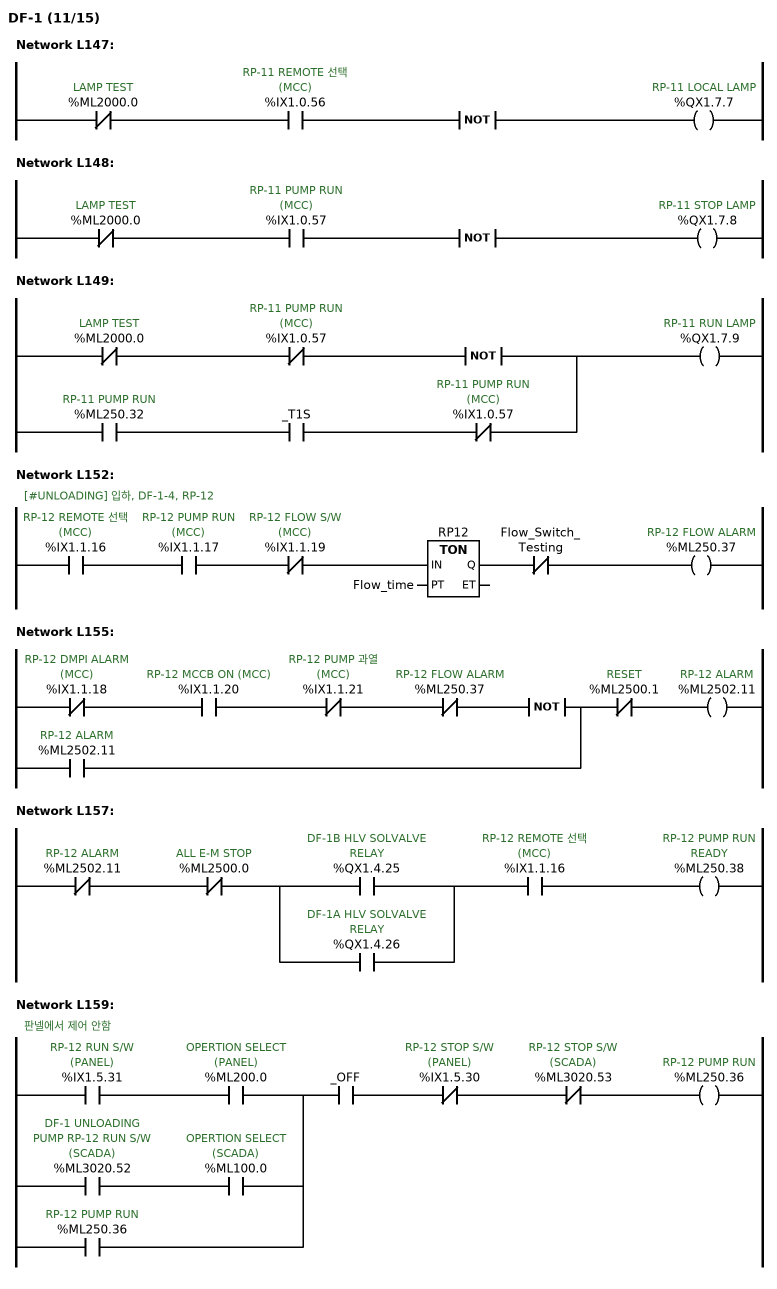
(* Rung L147 *)
%QX1.7.7 := NOT (NOT %ML2000.0 AND %IX1.0.56);
(* Rung L148 *)
%QX1.7.8 := NOT (NOT %ML2000.0 AND %IX1.0.57);
(* Rung L149 *)
%QX1.7.9 := NOT (NOT %ML2000.0 AND NOT %IX1.0.57) OR (%ML250.32 AND _T1S AND NOT %IX1.0.57);
(* [#UNLOADING] 입하, DF-1-4, RP-12 *)
(* Rung L152 *)
RP12(IN := %IX1.1.16 AND %IX1.1.17 AND NOT %IX1.1.19, PT := Flow_time);
%ML250.37 := RP12.Q AND NOT Flow_Switch_Testing;
(* Rung L155 *)
%ML2502.11 := (NOT (NOT %IX1.1.18 AND %IX1.1.20 AND NOT %IX1.1.21 AND NOT %ML250.37) OR %ML2502.11) AND NOT %ML2500.1;
(* Rung L157 *)
%ML250.38 := NOT %ML2502.11 AND NOT %ML2500.0 AND (%QX1.4.25 OR %QX1.4.26) AND %IX1.1.16;
(* Rung L159 *)
%ML250.36 := ((%IX1.5.31 AND %ML200.0) OR (%ML3020.52 AND %ML100.0) OR %ML250.36) AND _OFF AND NOT %IX1.5.30 AND NOT %ML3020.53;
(* 판넬에서 제어 안함 *)

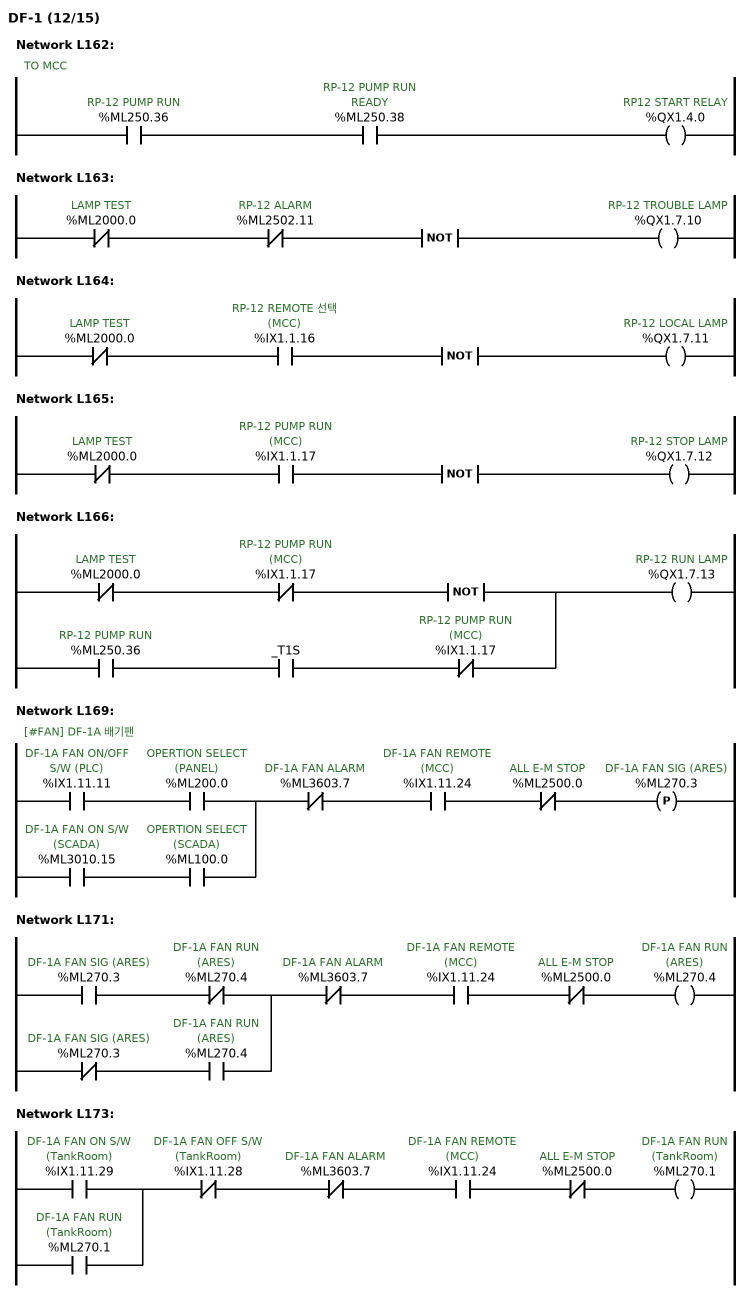
(* Rung L162 *)
%QX1.4.0 := %ML250.36 AND %ML250.38;
(* TO MCC *)
(* Rung L163 *)
%QX1.7.10 := NOT (NOT %ML2000.0 AND NOT %ML2502.11);
(* Rung L164 *)
%QX1.7.11 := NOT (NOT %ML2000.0 AND %IX1.1.16);
(* Rung L165 *)
%QX1.7.12 := NOT (NOT %ML2000.0 AND %IX1.1.17);
(* Rung L166 *)
%QX1.7.13 := NOT (NOT %ML2000.0 AND NOT %IX1.1.17) OR (%ML250.36 AND _T1S AND NOT %IX1.1.17);
(* [#FAN] DF-1A 배기팬 *)
(* Rung L169 *)
_e1(CLK := ((%IX1.11.11 AND %ML200.0) OR (%ML3010.15 AND %ML100.0)) AND NOT %ML3603.7 AND %IX1.11.24 AND NOT %ML2500.0);
%ML270.3 := _e1.Q;
(* Rung L171 *)
%ML270.4 := ((%ML270.3 AND NOT %ML270.4) OR (NOT %ML270.3 AND %ML270.4)) AND NOT %ML3603.7 AND %IX1.11.24 AND NOT %ML2500.0;
(* Rung L173 *)
%ML270.1 := (%IX1.11.29 OR %ML270.1) AND NOT %IX1.11.28 AND NOT %ML3603.7 AND %IX1.11.24 AND NOT %ML2500.0;

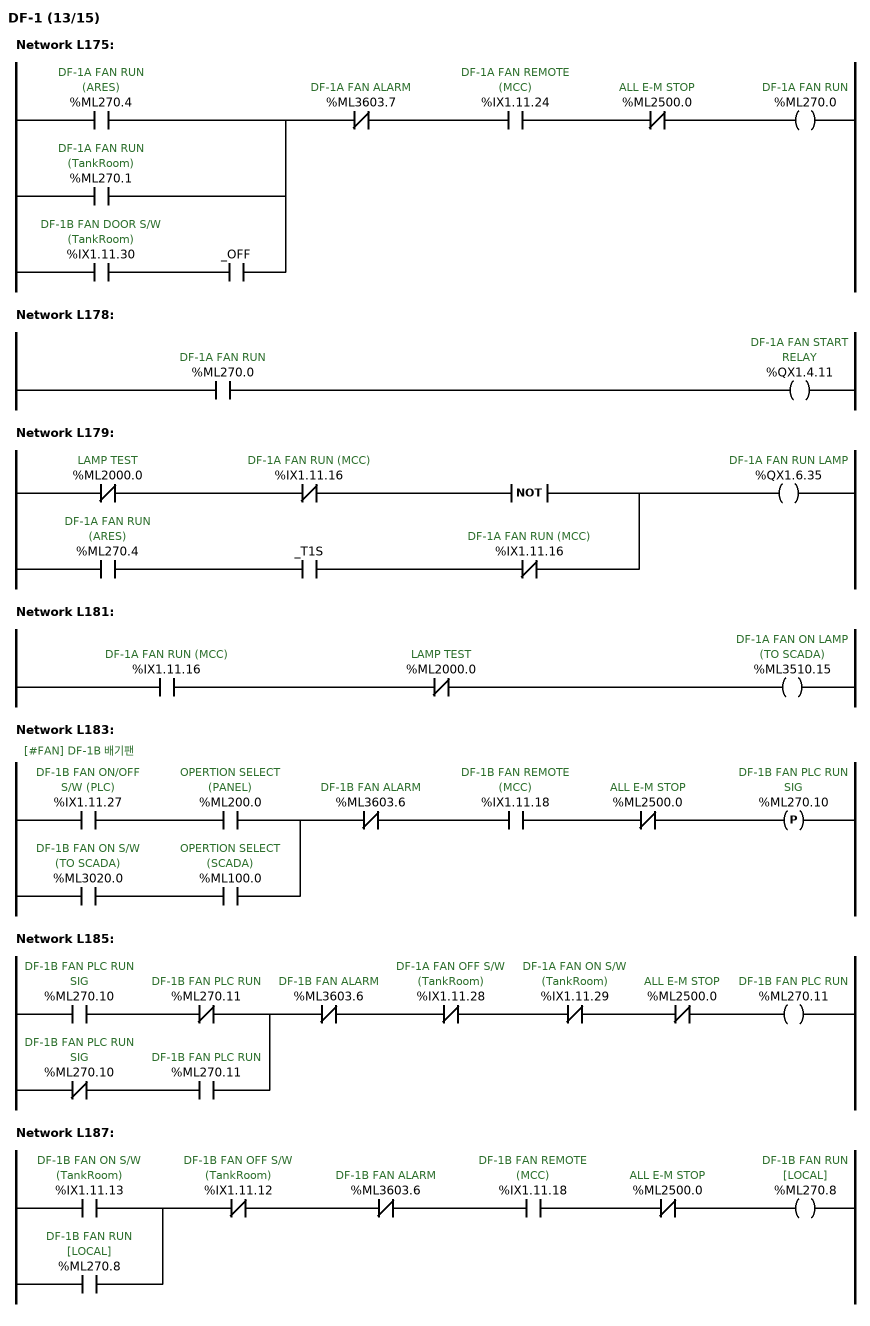
(* Rung L175 *)
%ML270.0 := (%ML270.4 OR %ML270.1 OR (%IX1.11.30 AND _OFF)) AND NOT %ML3603.7 AND %IX1.11.24 AND NOT %ML2500.0;
(* Rung L178 *)
%QX1.4.11 := %ML270.0;
(* Rung L179 *)
%QX1.6.35 := NOT (NOT %ML2000.0 AND NOT %IX1.11.16) OR (%ML270.4 AND _T1S AND NOT %IX1.11.16);
(* Rung L181 *)
%ML3510.15 := %IX1.11.16 AND NOT %ML2000.0;
(* [#FAN] DF-1B 배기팬 *)
(* Rung L183 *)
_e2(CLK := ((%IX1.11.27 AND %ML200.0) OR (%ML3020.0 AND %ML100.0)) AND NOT %ML3603.6 AND %IX1.11.18 AND NOT %ML2500.0);
%ML270.10 := _e2.Q;
(* Rung L185 *)
%ML270.11 := ((%ML270.10 AND NOT %ML270.11) OR (NOT %ML270.10 AND %ML270.11)) AND NOT %ML3603.6 AND NOT %IX1.11.28 AND NOT %IX1.11.29 AND NOT %ML2500.0;
(* Rung L187 *)
%ML270.8 := (%IX1.11.13 OR %ML270.8) AND NOT %IX1.11.12 AND NOT %ML3603.6 AND %IX1.11.18 AND NOT %ML2500.0;

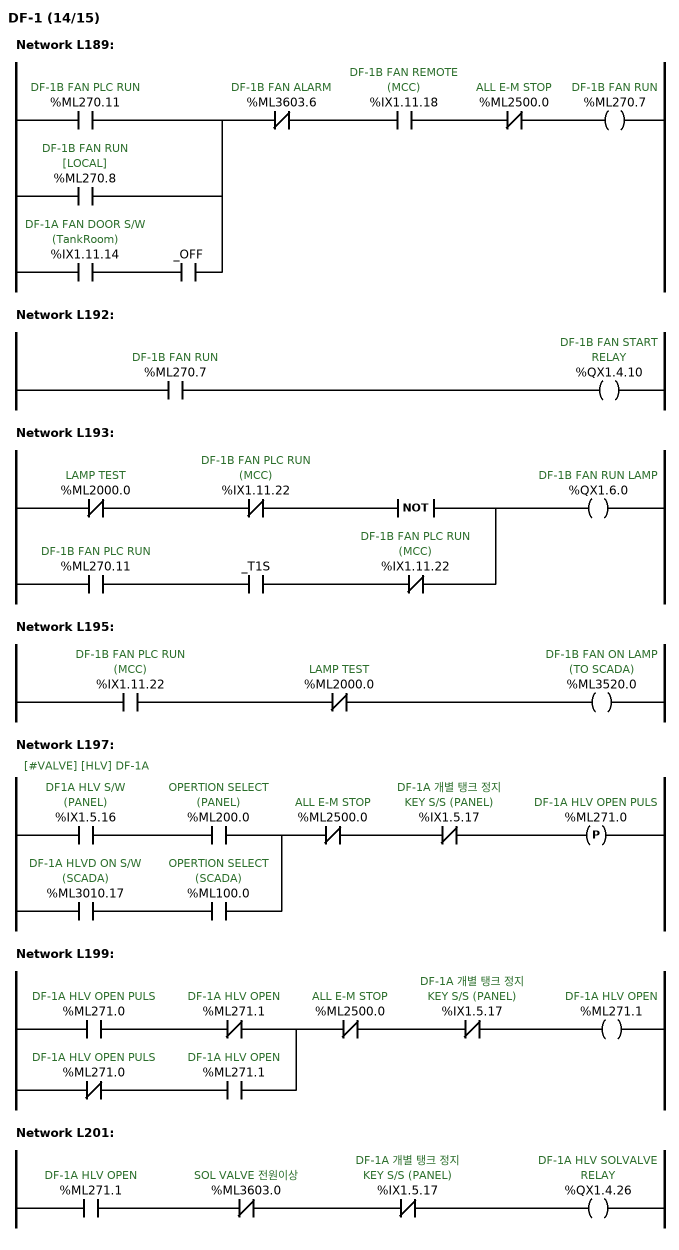
(* Rung L189 *)
%ML270.7 := (%ML270.11 OR %ML270.8 OR (%IX1.11.14 AND _OFF)) AND NOT %ML3603.6 AND %IX1.11.18 AND NOT %ML2500.0;
(* Rung L192 *)
%QX1.4.10 := %ML270.7;
(* Rung L193 *)
%QX1.6.0 := NOT (NOT %ML2000.0 AND NOT %IX1.11.22) OR (%ML270.11 AND _T1S AND NOT %IX1.11.22);
(* Rung L195 *)
%ML3520.0 := %IX1.11.22 AND NOT %ML2000.0;
(* [#VALVE] [HLV] DF-1A *)
(* Rung L197 *)
_e3(CLK := ((%IX1.5.16 AND %ML200.0) OR (%ML3010.17 AND %ML100.0)) AND NOT %ML2500.0 AND NOT %IX1.5.17);
%ML271.0 := _e3.Q;
(* Rung L199 *)
%ML271.1 := ((%ML271.0 AND NOT %ML271.1) OR (NOT %ML271.0 AND %ML271.1)) AND NOT %ML2500.0 AND NOT %IX1.5.17;
(* Rung L201 *)
%QX1.4.26 := %ML271.1 AND NOT %ML3603.0 AND NOT %IX1.5.17;

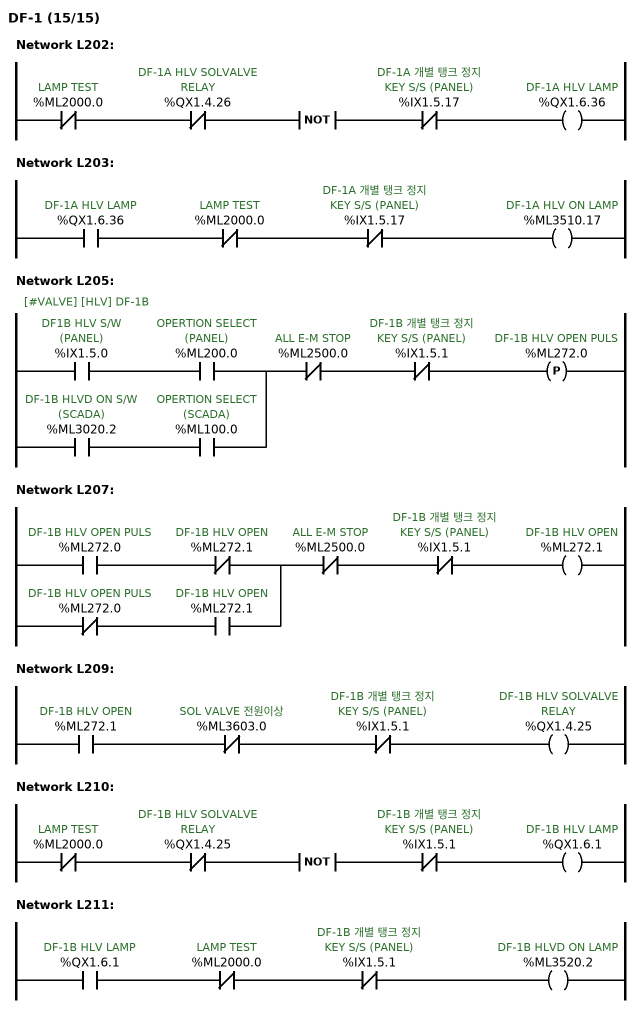
(* Rung L202 *)
%QX1.6.36 := NOT (NOT %ML2000.0 AND NOT %QX1.4.26) AND NOT %IX1.5.17;
(* Rung L203 *)
%ML3510.17 := %QX1.6.36 AND NOT %ML2000.0 AND NOT %IX1.5.17;
(* [#VALVE] [HLV] DF-1B *)
(* Rung L205 *)
_e4(CLK := ((%IX1.5.0 AND %ML200.0) OR (%ML3020.2 AND %ML100.0)) AND NOT %ML2500.0 AND NOT %IX1.5.1);
%ML272.0 := _e4.Q;
(* Rung L207 *)
%ML272.1 := ((%ML272.0 AND NOT %ML272.1) OR (NOT %ML272.0 AND %ML272.1)) AND NOT %ML2500.0 AND NOT %IX1.5.1;
(* Rung L209 *)
%QX1.4.25 := %ML272.1 AND NOT %ML3603.0 AND NOT %IX1.5.1;
(* Rung L210 *)
%QX1.6.1 := NOT (NOT %ML2000.0 AND NOT %QX1.4.25) AND NOT %IX1.5.1;
(* Rung L211 *)
%ML3520.2 := %QX1.6.1 AND NOT %ML2000.0 AND NOT %IX1.5.1;
END_PROGRAM

PROGRAM DF-M (* task: 스캔 프로그램 *)
VAR_EXTERNAL
    Flow_Switch_Testing : BOOL;
    Flow_time : TIME;
END_VAR
VAR
    RP10 : TON;
    RP11 : TON;
    RP12 : TON;
    RP13 : TON;
    RP14 : TON;
    RP15 : TON;
    RP16 : TON;
    RP17 : TON;
    RP18 : TON;
    RP7 : TON;
    RP8 : TON;
    RP9 : TON;
    SUMP02 : TON; (* SP-2 *)
    SUMP04 : TON;
END_VAR
VAR
    _t1 : BOOL;
    _t2 : BOOL;
    _t3 : BOOL;
    _t4 : BOOL;
    _e5 : R_TRIG;
END_VAR

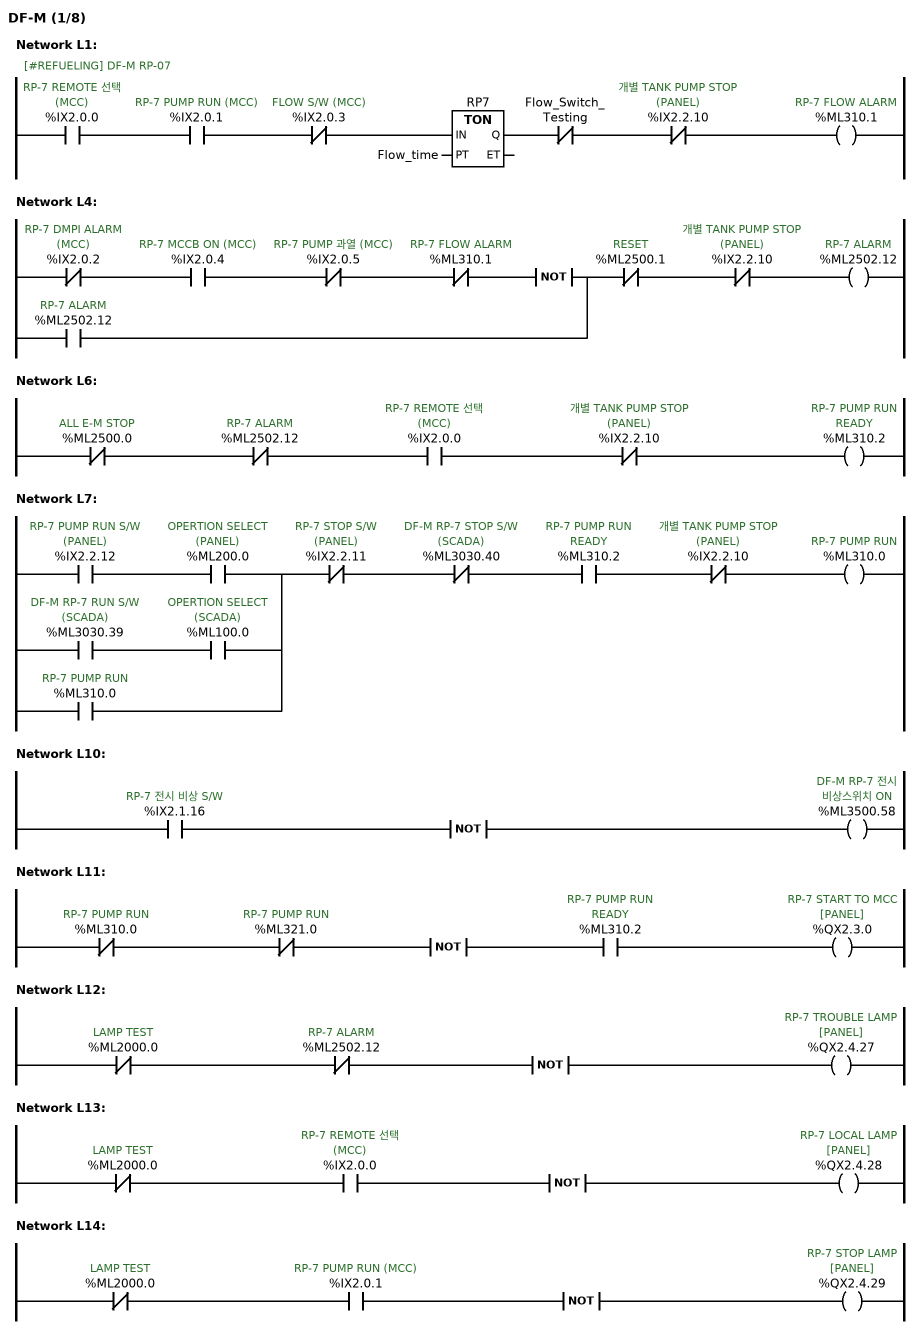
(* [#REFUELING] DF-M RP-07 *)
(* Rung L1 *)
RP7(IN := %IX2.0.0 AND %IX2.0.1 AND NOT %IX2.0.3, PT := Flow_time);
%ML310.1 := RP7.Q AND NOT Flow_Switch_Testing AND NOT %IX2.2.10;
(* Rung L4 *)
%ML2502.12 := (NOT (NOT %IX2.0.2 AND %IX2.0.4 AND NOT %IX2.0.5 AND NOT %ML310.1) OR %ML2502.12) AND NOT %ML2500.1 AND NOT %IX2.2.10;
(* Rung L6 *)
%ML310.2 := NOT %ML2500.0 AND NOT %ML2502.12 AND %IX2.0.0 AND NOT %IX2.2.10;
(* Rung L7 *)
%ML310.0 := ((%IX2.2.12 AND %ML200.0) OR (%ML3030.39 AND %ML100.0) OR %ML310.0) AND NOT %IX2.2.11 AND NOT %ML3030.40 AND %ML310.2 AND NOT %IX2.2.10;
(* Rung L10 *)
%ML3500.58 := NOT %IX2.1.16;
(* Rung L11 *)
%QX2.3.0 := NOT (NOT %ML310.0 AND NOT %ML321.0) AND %ML310.2;
(* Rung L12 *)
%QX2.4.27 := NOT (NOT %ML2000.0 AND NOT %ML2502.12);
(* Rung L13 *)
%QX2.4.28 := NOT (NOT %ML2000.0 AND %IX2.0.0);
(* Rung L14 *)
%QX2.4.29 := NOT (NOT %ML2000.0 AND %IX2.0.1);

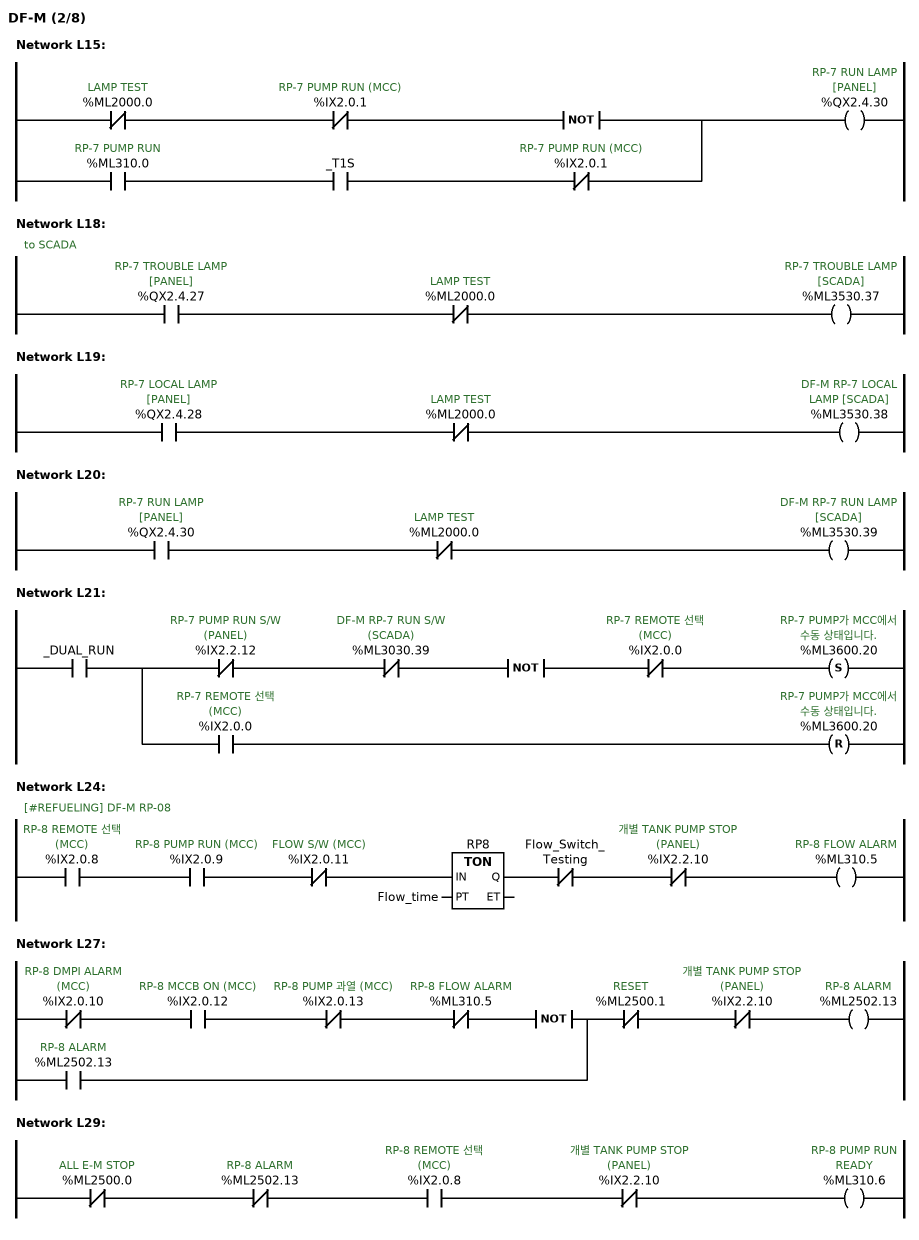
(* Rung L15 *)
%QX2.4.30 := NOT (NOT %ML2000.0 AND NOT %IX2.0.1) OR (%ML310.0 AND _T1S AND NOT %IX2.0.1);
(* to SCADA *)
(* Rung L18 *)
%ML3530.37 := %QX2.4.27 AND NOT %ML2000.0;
(* Rung L19 *)
%ML3530.38 := %QX2.4.28 AND NOT %ML2000.0;
(* Rung L20 *)
%ML3530.39 := %QX2.4.30 AND NOT %ML2000.0;
(* Rung L21 *)
IF NOT (_DUAL_RUN AND NOT %IX2.2.12 AND NOT %ML3030.39) AND NOT %IX2.0.0 THEN %ML3600.20 := TRUE; END_IF;
IF _DUAL_RUN AND %IX2.0.0 THEN %ML3600.20 := FALSE; END_IF;
(* [#REFUELING] DF-M RP-08 *)
(* Rung L24 *)
RP8(IN := %IX2.0.8 AND %IX2.0.9 AND NOT %IX2.0.11, PT := Flow_time);
%ML310.5 := RP8.Q AND NOT Flow_Switch_Testing AND NOT %IX2.2.10;
(* Rung L27 *)
%ML2502.13 := (NOT (NOT %IX2.0.10 AND %IX2.0.12 AND NOT %IX2.0.13 AND NOT %ML310.5) OR %ML2502.13) AND NOT %ML2500.1 AND NOT %IX2.2.10;
(* Rung L29 *)
%ML310.6 := NOT %ML2500.0 AND NOT %ML2502.13 AND %IX2.0.8 AND NOT %IX2.2.10;

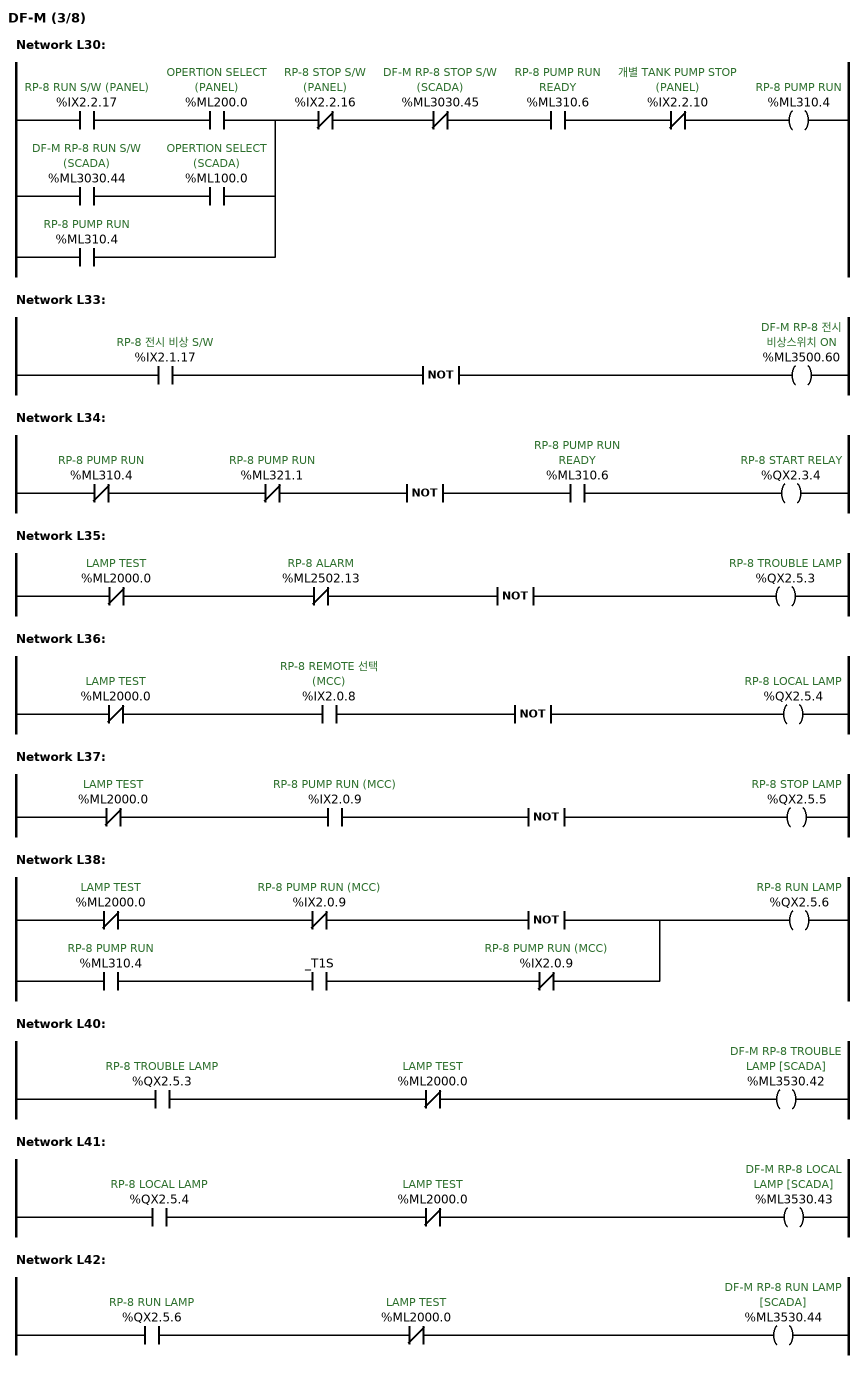
(* Rung L30 *)
%ML310.4 := ((%IX2.2.17 AND %ML200.0) OR (%ML3030.44 AND %ML100.0) OR %ML310.4) AND NOT %IX2.2.16 AND NOT %ML3030.45 AND %ML310.6 AND NOT %IX2.2.10;
(* Rung L33 *)
%ML3500.60 := NOT %IX2.1.17;
(* Rung L34 *)
%QX2.3.4 := NOT (NOT %ML310.4 AND NOT %ML321.1) AND %ML310.6;
(* Rung L35 *)
%QX2.5.3 := NOT (NOT %ML2000.0 AND NOT %ML2502.13);
(* Rung L36 *)
%QX2.5.4 := NOT (NOT %ML2000.0 AND %IX2.0.8);
(* Rung L37 *)
%QX2.5.5 := NOT (NOT %ML2000.0 AND %IX2.0.9);
(* Rung L38 *)
%QX2.5.6 := NOT (NOT %ML2000.0 AND NOT %IX2.0.9) OR (%ML310.4 AND _T1S AND NOT %IX2.0.9);
(* Rung L40 *)
%ML3530.42 := %QX2.5.3 AND NOT %ML2000.0;
(* Rung L41 *)
%ML3530.43 := %QX2.5.4 AND NOT %ML2000.0;
(* Rung L42 *)
%ML3530.44 := %QX2.5.6 AND NOT %ML2000.0;

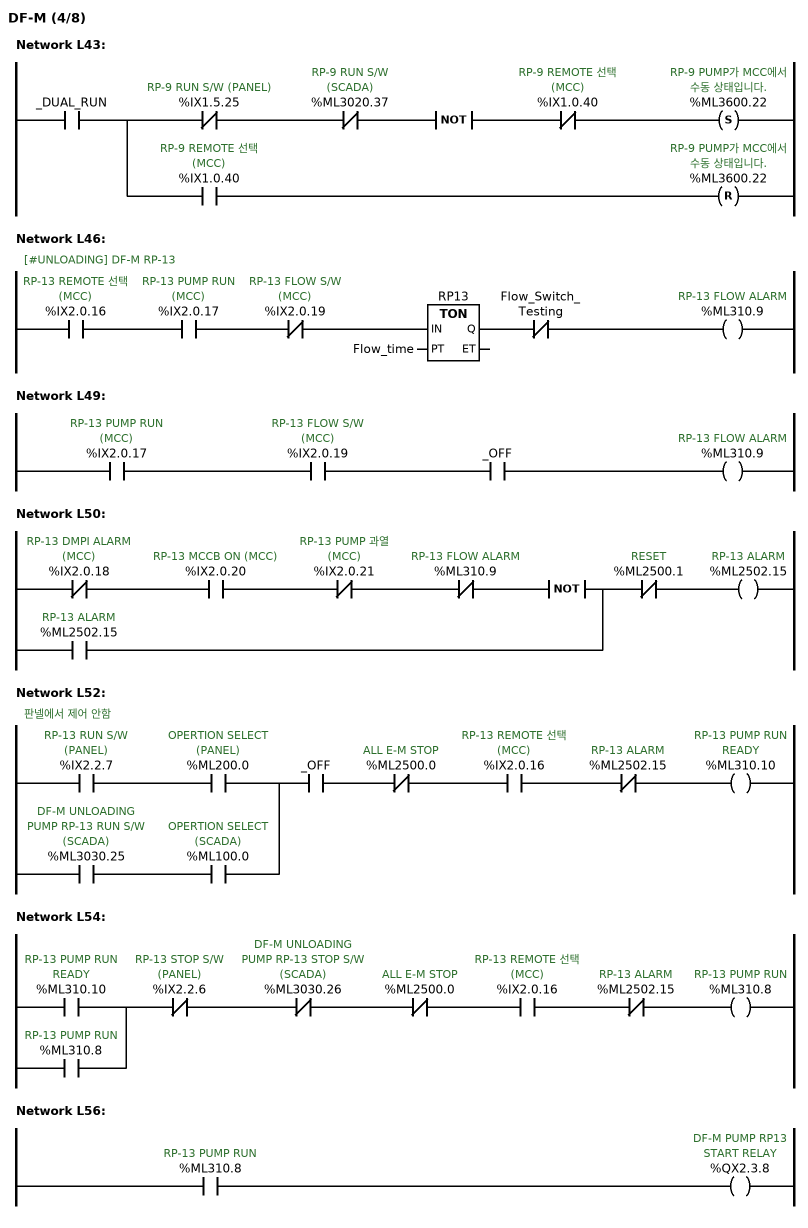
(* Rung L43 *)
IF NOT (_DUAL_RUN AND NOT %IX1.5.25 AND NOT %ML3020.37) AND NOT %IX1.0.40 THEN %ML3600.22 := TRUE; END_IF;
IF _DUAL_RUN AND %IX1.0.40 THEN %ML3600.22 := FALSE; END_IF;
(* [#UNLOADING] DF-M RP-13 *)
(* Rung L46 *)
RP13(IN := %IX2.0.16 AND %IX2.0.17 AND NOT %IX2.0.19, PT := Flow_time);
%ML310.9 := RP13.Q AND NOT Flow_Switch_Testing;
(* Rung L49 *)
%ML310.9 := %IX2.0.17 AND %IX2.0.19 AND _OFF;
(* Rung L50 *)
%ML2502.15 := (NOT (NOT %IX2.0.18 AND %IX2.0.20 AND NOT %IX2.0.21 AND NOT %ML310.9) OR %ML2502.15) AND NOT %ML2500.1;
(* Rung L52 *)
%ML310.10 := ((%IX2.2.7 AND %ML200.0) OR (%ML3030.25 AND %ML100.0)) AND _OFF AND NOT %ML2500.0 AND %IX2.0.16 AND NOT %ML2502.15;
(* 판넬에서 제어 안함 *)
(* Rung L54 *)
%ML310.8 := (%ML310.10 OR %ML310.8) AND NOT %IX2.2.6 AND NOT %ML3030.26 AND NOT %ML2500.0 AND %IX2.0.16 AND NOT %ML2502.15;
(* Rung L56 *)
%QX2.3.8 := %ML310.8;

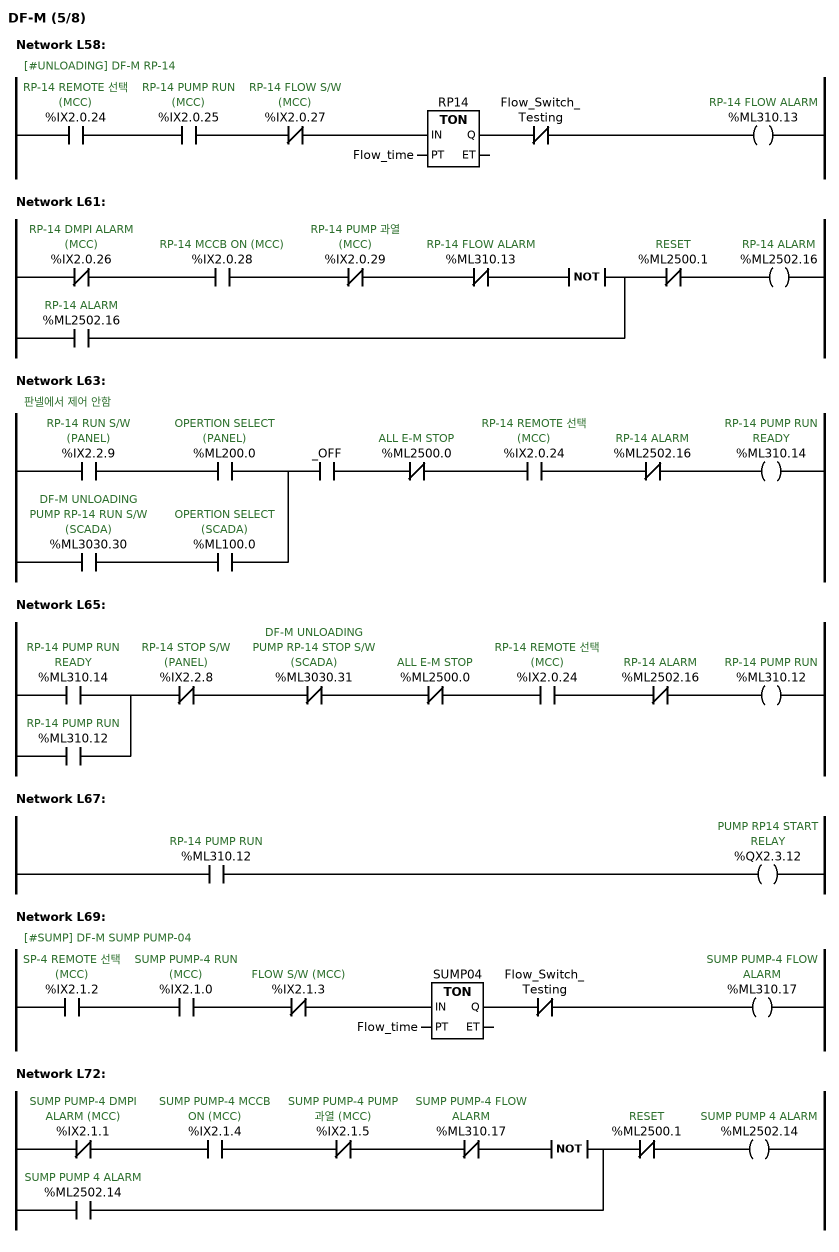
(* [#UNLOADING] DF-M RP-14 *)
(* Rung L58 *)
RP14(IN := %IX2.0.24 AND %IX2.0.25 AND NOT %IX2.0.27, PT := Flow_time);
%ML310.13 := RP14.Q AND NOT Flow_Switch_Testing;
(* Rung L61 *)
%ML2502.16 := (NOT (NOT %IX2.0.26 AND %IX2.0.28 AND NOT %IX2.0.29 AND NOT %ML310.13) OR %ML2502.16) AND NOT %ML2500.1;
(* Rung L63 *)
%ML310.14 := ((%IX2.2.9 AND %ML200.0) OR (%ML3030.30 AND %ML100.0)) AND _OFF AND NOT %ML2500.0 AND %IX2.0.24 AND NOT %ML2502.16;
(* 판넬에서 제어 안함 *)
(* Rung L65 *)
%ML310.12 := (%ML310.14 OR %ML310.12) AND NOT %IX2.2.8 AND NOT %ML3030.31 AND NOT %ML2500.0 AND %IX2.0.24 AND NOT %ML2502.16;
(* Rung L67 *)
%QX2.3.12 := %ML310.12;
(* [#SUMP] DF-M SUMP PUMP-04 *)
(* Rung L69 *)
SUMP04(IN := %IX2.1.2 AND %IX2.1.0 AND NOT %IX2.1.3, PT := Flow_time);
%ML310.17 := SUMP04.Q AND NOT Flow_Switch_Testing;
(* Rung L72 *)
%ML2502.14 := (NOT (NOT %IX2.1.1 AND %IX2.1.4 AND NOT %IX2.1.5 AND NOT %ML310.17) OR %ML2502.14) AND NOT %ML2500.1;

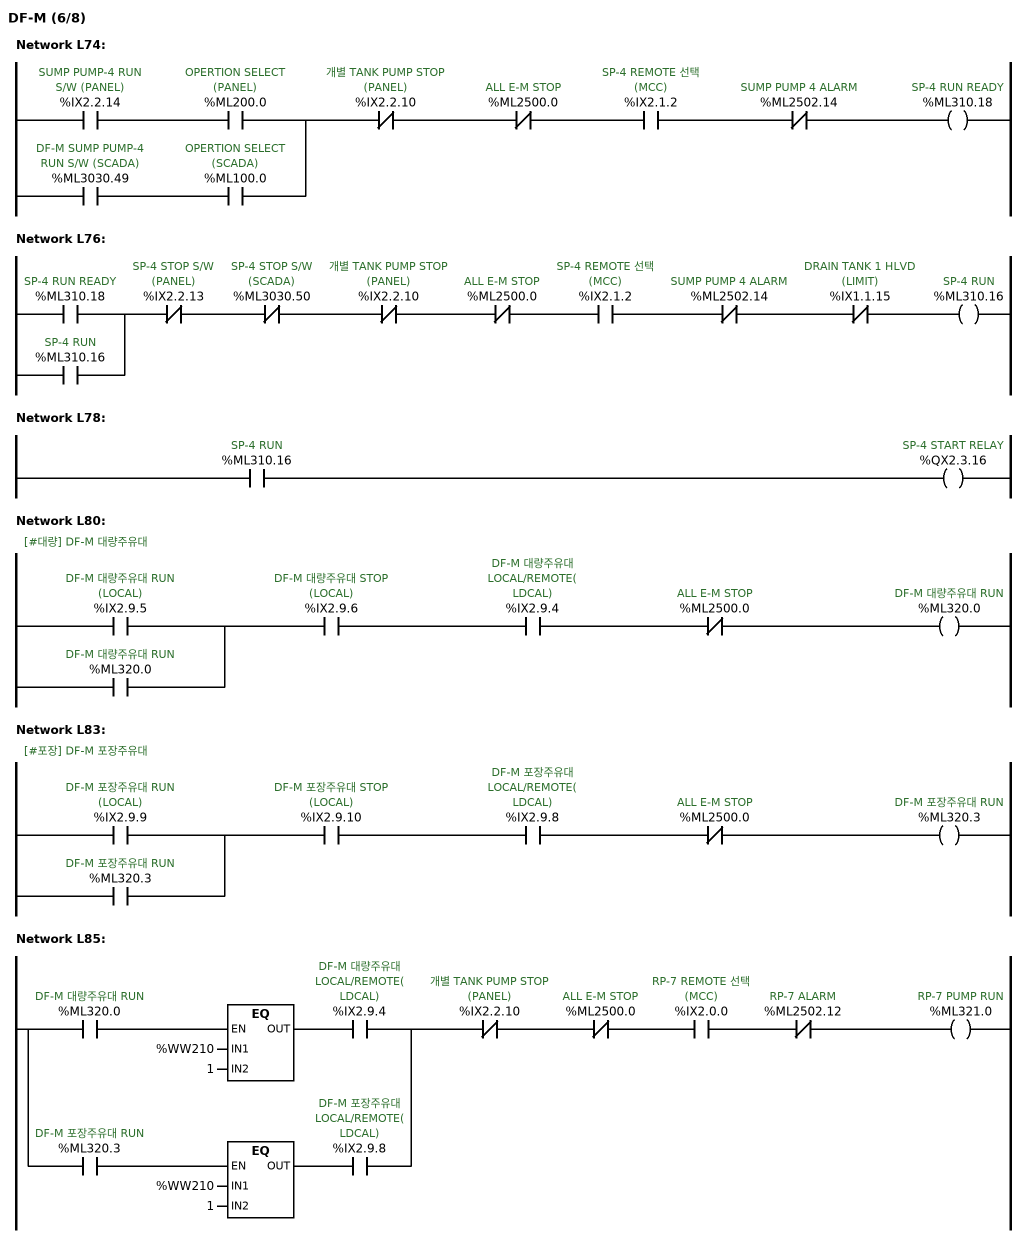
(* Rung L74 *)
%ML310.18 := ((%IX2.2.14 AND %ML200.0) OR (%ML3030.49 AND %ML100.0)) AND NOT %IX2.2.10 AND NOT %ML2500.0 AND %IX2.1.2 AND NOT %ML2502.14;
(* Rung L76 *)
%ML310.16 := (%ML310.18 OR %ML310.16) AND NOT %IX2.2.13 AND NOT %ML3030.50 AND NOT %IX2.2.10 AND NOT %ML2500.0 AND %IX2.1.2 AND NOT %ML2502.14 AND NOT %IX1.1.15;
(* Rung L78 *)
%QX2.3.16 := %ML310.16;
(* [#대량] DF-M 대량주유대 *)
(* Rung L80 *)
%ML320.0 := (%IX2.9.5 OR %ML320.0) AND %IX2.9.6 AND %IX2.9.4 AND NOT %ML2500.0;
(* [#포장] DF-M 포장주유대 *)
(* Rung L83 *)
%ML320.3 := (%IX2.9.9 OR %ML320.3) AND %IX2.9.10 AND %IX2.9.8 AND NOT %ML2500.0;
(* Rung L85 *)
IF %ML320.0 THEN _t1 := %WW210 = 1; END_IF;
IF %ML320.3 THEN _t2 := %WW210 = 1; END_IF;
%ML321.0 := ((_t1 AND %IX2.9.4) OR (_t2 AND %IX2.9.8)) AND NOT %IX2.2.10 AND NOT %ML2500.0 AND %IX2.0.0 AND NOT %ML2502.12;

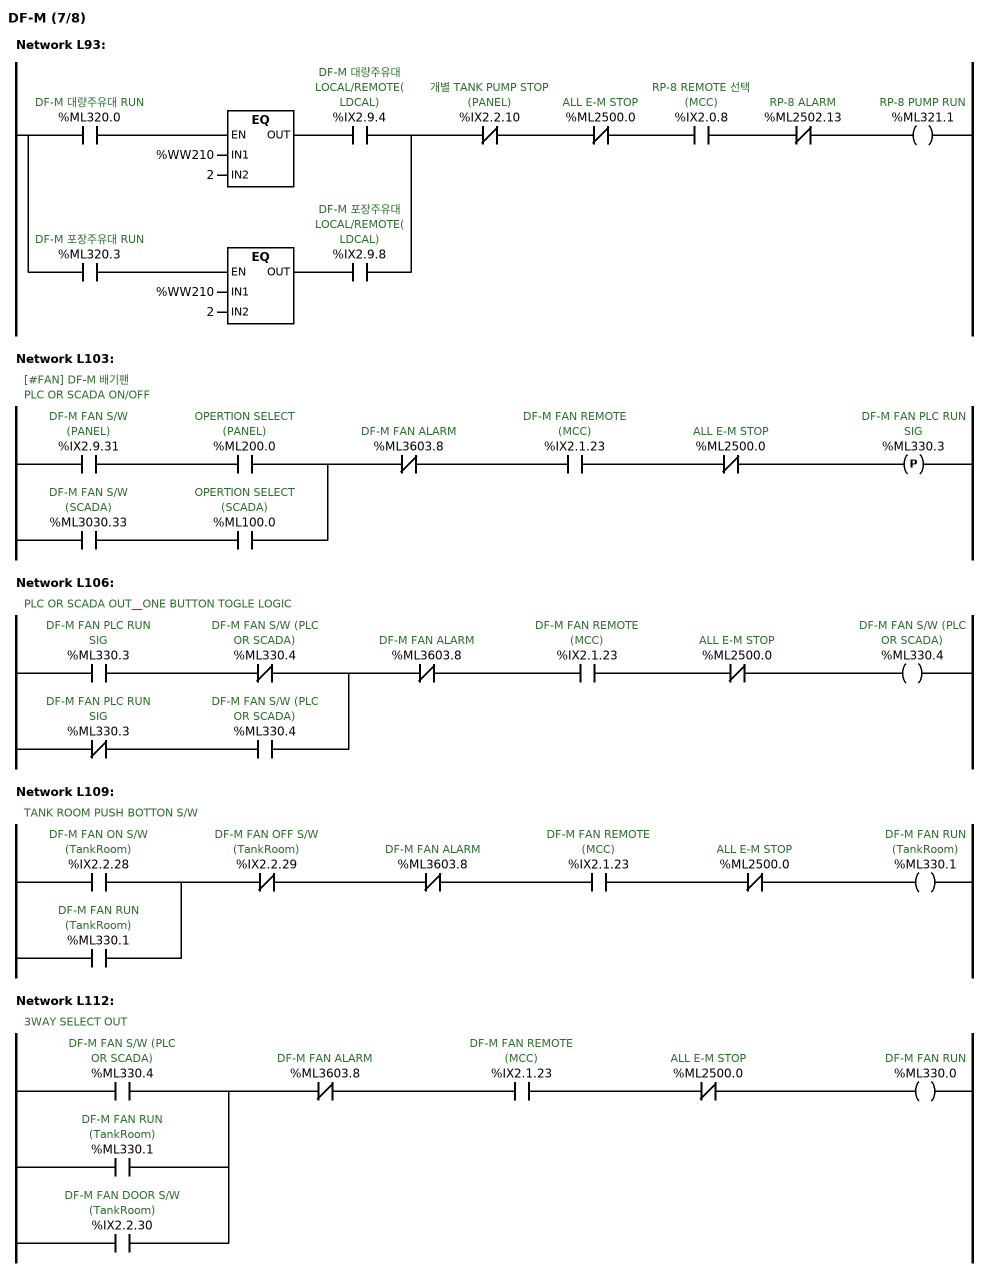
(* Rung L93 *)
IF %ML320.0 THEN _t3 := %WW210 = 2; END_IF;
IF %ML320.3 THEN _t4 := %WW210 = 2; END_IF;
%ML321.1 := ((_t3 AND %IX2.9.4) OR (_t4 AND %IX2.9.8)) AND NOT %IX2.2.10 AND NOT %ML2500.0 AND %IX2.0.8 AND NOT %ML2502.13;
(* [#FAN] DF-M 배기팬 *)
(* PLC OR SCADA ON/OFF *)
(* Rung L103 *)
_e5(CLK := ((%IX2.9.31 AND %ML200.0) OR (%ML3030.33 AND %ML100.0)) AND NOT %ML3603.8 AND %IX2.1.23 AND NOT %ML2500.0);
%ML330.3 := _e5.Q;
(* PLC OR SCADA OUT__ONE BUTTON TOGLE LOGIC *)
(* Rung L106 *)
%ML330.4 := ((%ML330.3 AND NOT %ML330.4) OR (NOT %ML330.3 AND %ML330.4)) AND NOT %ML3603.8 AND %IX2.1.23 AND NOT %ML2500.0;
(* TANK ROOM PUSH BOTTON S/W *)
(* Rung L109 *)
%ML330.1 := (%IX2.2.28 OR %ML330.1) AND NOT %IX2.2.29 AND NOT %ML3603.8 AND %IX2.1.23 AND NOT %ML2500.0;
(* 3WAY SELECT OUT *)
(* Rung L112 *)
%ML330.0 := (%ML330.4 OR %ML330.1 OR %IX2.2.30) AND NOT %ML3603.8 AND %IX2.1.23 AND NOT %ML2500.0;

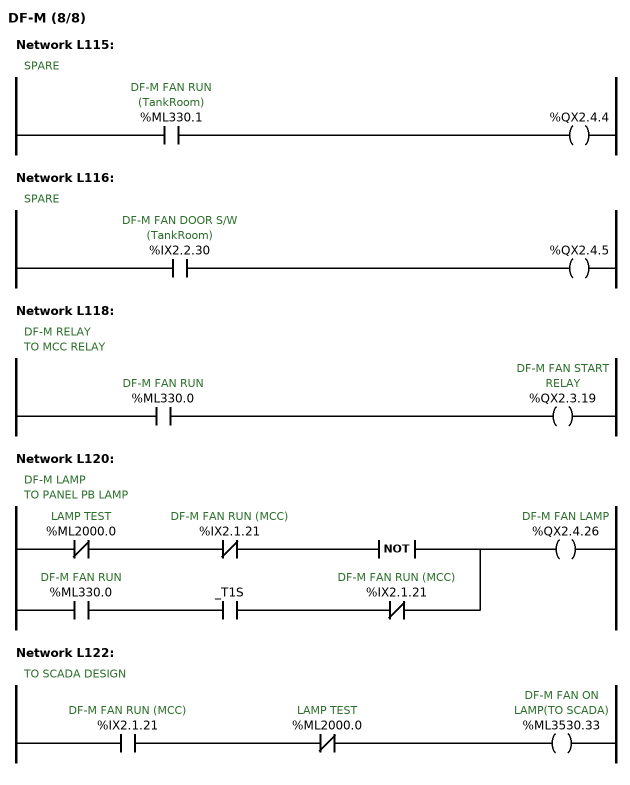
(* Rung L115 *)
%QX2.4.4 := %ML330.1;
(* SPARE *)
(* Rung L116 *)
%QX2.4.5 := %IX2.2.30;
(* SPARE *)
(* DF-M RELAY *)
(* Rung L118 *)
%QX2.3.19 := %ML330.0;
(* TO MCC RELAY *)
(* DF-M LAMP *)
(* Rung L120 *)
%QX2.4.26 := NOT (NOT %ML2000.0 AND NOT %IX2.1.21) OR (%ML330.0 AND _T1S AND NOT %IX2.1.21);
(* TO PANEL PB LAMP *)
(* Rung L122 *)
%ML3530.33 := %IX2.1.21 AND NOT %ML2000.0;
(* TO SCADA DESIGN *)
END_PROGRAM

PROGRAM MOGAS (* task: 스캔 프로그램 *)
VAR
    DP01 : TON; (* DRAIN PUMP FLOW SENSOR *)
    RP10 : TON;
    RP11 : TON;
    RP12 : TON;
    RP13 : TON;
    RP14 : TON;
    RP15 : TON;
    RP16 : TON;
    RP17 : TON;
    RP18 : TON;
    RP19 : TON;
    RP20 : TON;
    RP5 : TON;
    RP6 : TON;
    RP7 : TON;
    RP8 : TON;
    RP9 : TON;
    SUMP04 : TON;
END_VAR
VAR_EXTERNAL
    Flow_Switch_Testing : BOOL;
    Flow_time : TIME;
END_VAR
VAR
    _t1 : BOOL;
    _t2 : BOOL;
    _t3 : BOOL;
    _t4 : BOOL;
    _e5 : R_TRIG;
END_VAR

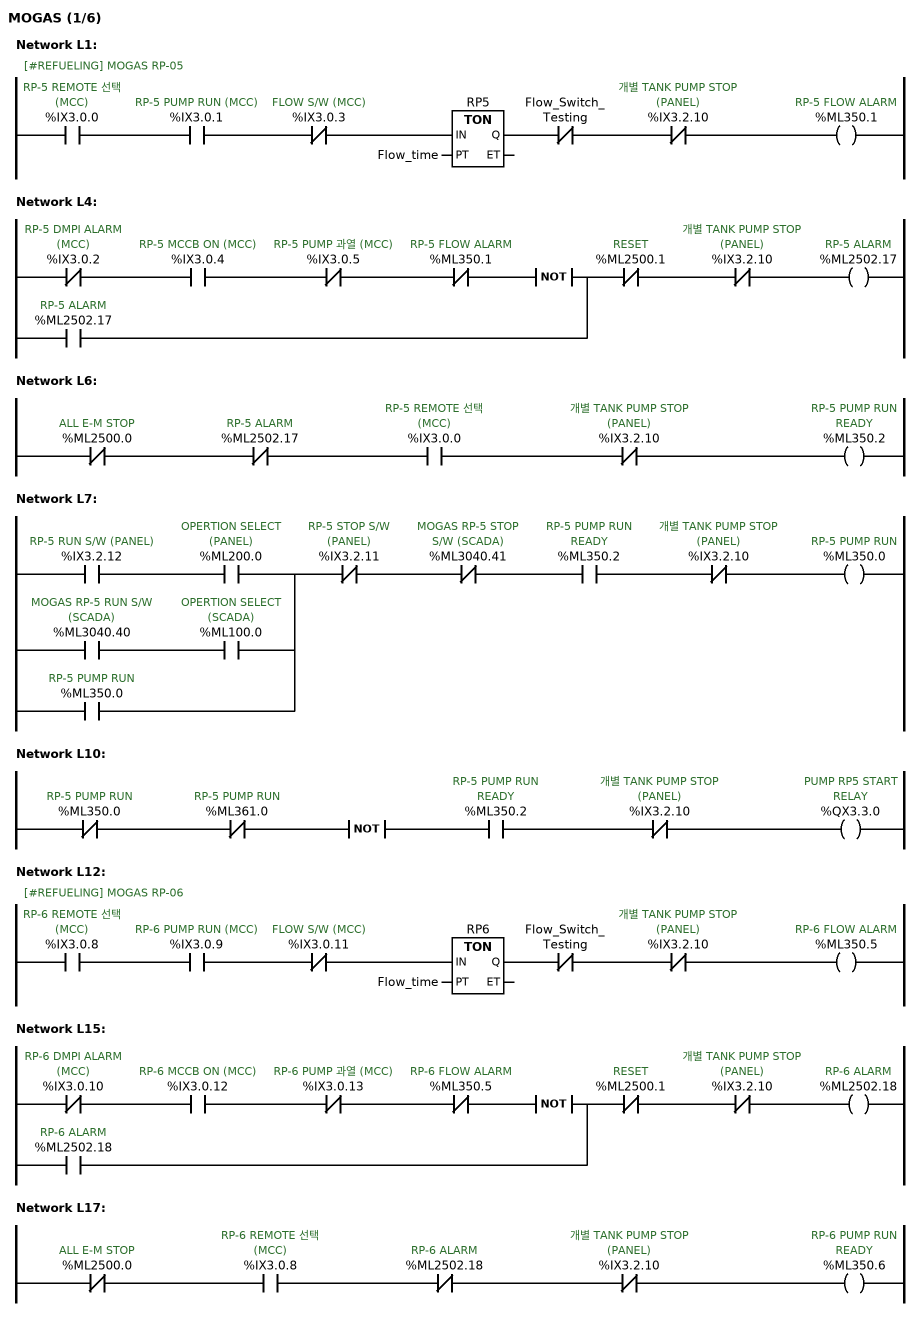
(* [#REFUELING] MOGAS RP-05 *)
(* Rung L1 *)
RP5(IN := %IX3.0.0 AND %IX3.0.1 AND NOT %IX3.0.3, PT := Flow_time);
%ML350.1 := RP5.Q AND NOT Flow_Switch_Testing AND NOT %IX3.2.10;
(* Rung L4 *)
%ML2502.17 := (NOT (NOT %IX3.0.2 AND %IX3.0.4 AND NOT %IX3.0.5 AND NOT %ML350.1) OR %ML2502.17) AND NOT %ML2500.1 AND NOT %IX3.2.10;
(* Rung L6 *)
%ML350.2 := NOT %ML2500.0 AND NOT %ML2502.17 AND %IX3.0.0 AND NOT %IX3.2.10;
(* Rung L7 *)
%ML350.0 := ((%IX3.2.12 AND %ML200.0) OR (%ML3040.40 AND %ML100.0) OR %ML350.0) AND NOT %IX3.2.11 AND NOT %ML3040.41 AND %ML350.2 AND NOT %IX3.2.10;
(* Rung L10 *)
%QX3.3.0 := NOT (NOT %ML350.0 AND NOT %ML361.0) AND %ML350.2 AND NOT %IX3.2.10;
(* [#REFUELING] MOGAS RP-06 *)
(* Rung L12 *)
RP6(IN := %IX3.0.8 AND %IX3.0.9 AND NOT %IX3.0.11, PT := Flow_time);
%ML350.5 := RP6.Q AND NOT Flow_Switch_Testing AND NOT %IX3.2.10;
(* Rung L15 *)
%ML2502.18 := (NOT (NOT %IX3.0.10 AND %IX3.0.12 AND NOT %IX3.0.13 AND NOT %ML350.5) OR %ML2502.18) AND NOT %ML2500.1 AND NOT %IX3.2.10;
(* Rung L17 *)
%ML350.6 := NOT %ML2500.0 AND %IX3.0.8 AND NOT %ML2502.18 AND NOT %IX3.2.10;

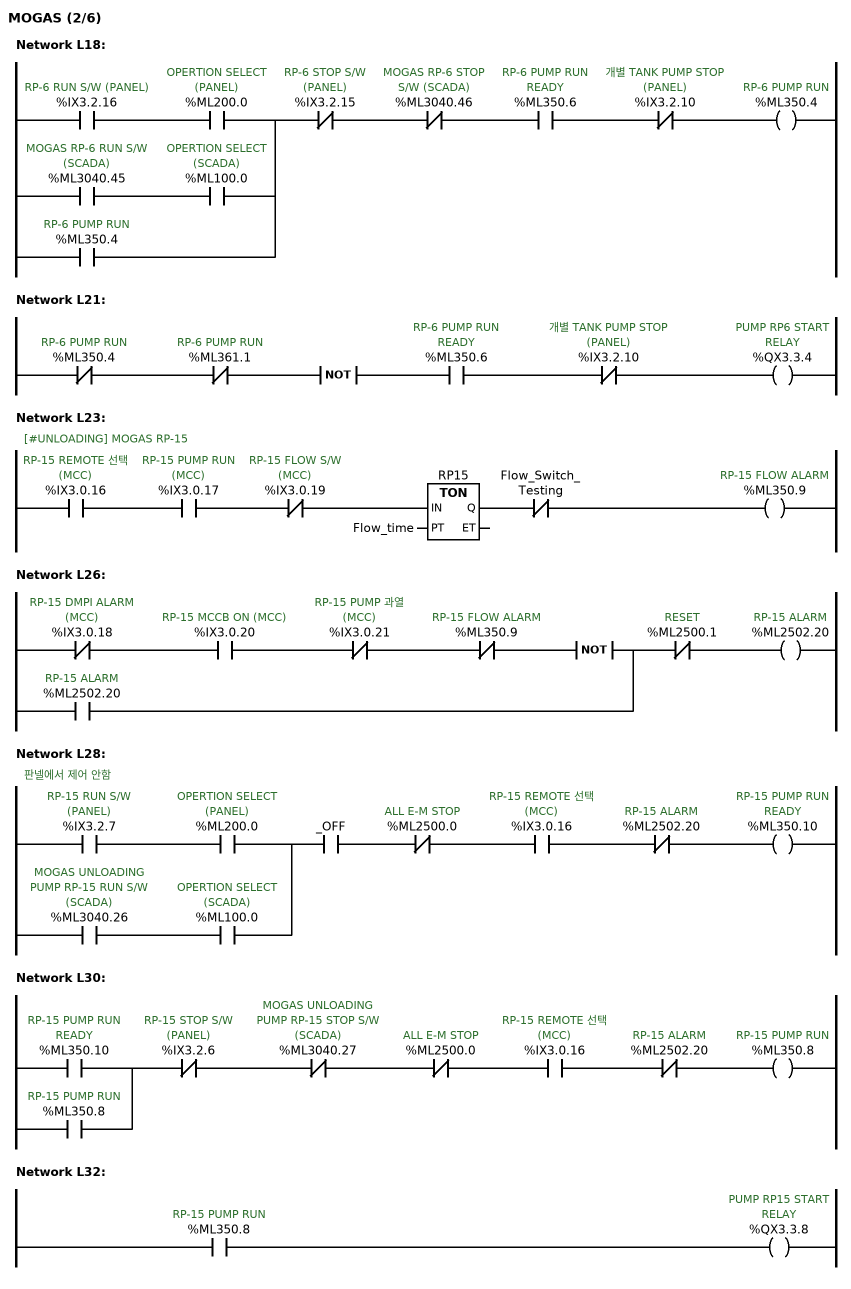
(* Rung L18 *)
%ML350.4 := ((%IX3.2.16 AND %ML200.0) OR (%ML3040.45 AND %ML100.0) OR %ML350.4) AND NOT %IX3.2.15 AND NOT %ML3040.46 AND %ML350.6 AND NOT %IX3.2.10;
(* Rung L21 *)
%QX3.3.4 := NOT (NOT %ML350.4 AND NOT %ML361.1) AND %ML350.6 AND NOT %IX3.2.10;
(* [#UNLOADING] MOGAS RP-15 *)
(* Rung L23 *)
RP15(IN := %IX3.0.16 AND %IX3.0.17 AND NOT %IX3.0.19, PT := Flow_time);
%ML350.9 := RP15.Q AND NOT Flow_Switch_Testing;
(* Rung L26 *)
%ML2502.20 := (NOT (NOT %IX3.0.18 AND %IX3.0.20 AND NOT %IX3.0.21 AND NOT %ML350.9) OR %ML2502.20) AND NOT %ML2500.1;
(* Rung L28 *)
%ML350.10 := ((%IX3.2.7 AND %ML200.0) OR (%ML3040.26 AND %ML100.0)) AND _OFF AND NOT %ML2500.0 AND %IX3.0.16 AND NOT %ML2502.20;
(* 판넬에서 제어 안함 *)
(* Rung L30 *)
%ML350.8 := (%ML350.10 OR %ML350.8) AND NOT %IX3.2.6 AND NOT %ML3040.27 AND NOT %ML2500.0 AND %IX3.0.16 AND NOT %ML2502.20;
(* Rung L32 *)
%QX3.3.8 := %ML350.8;

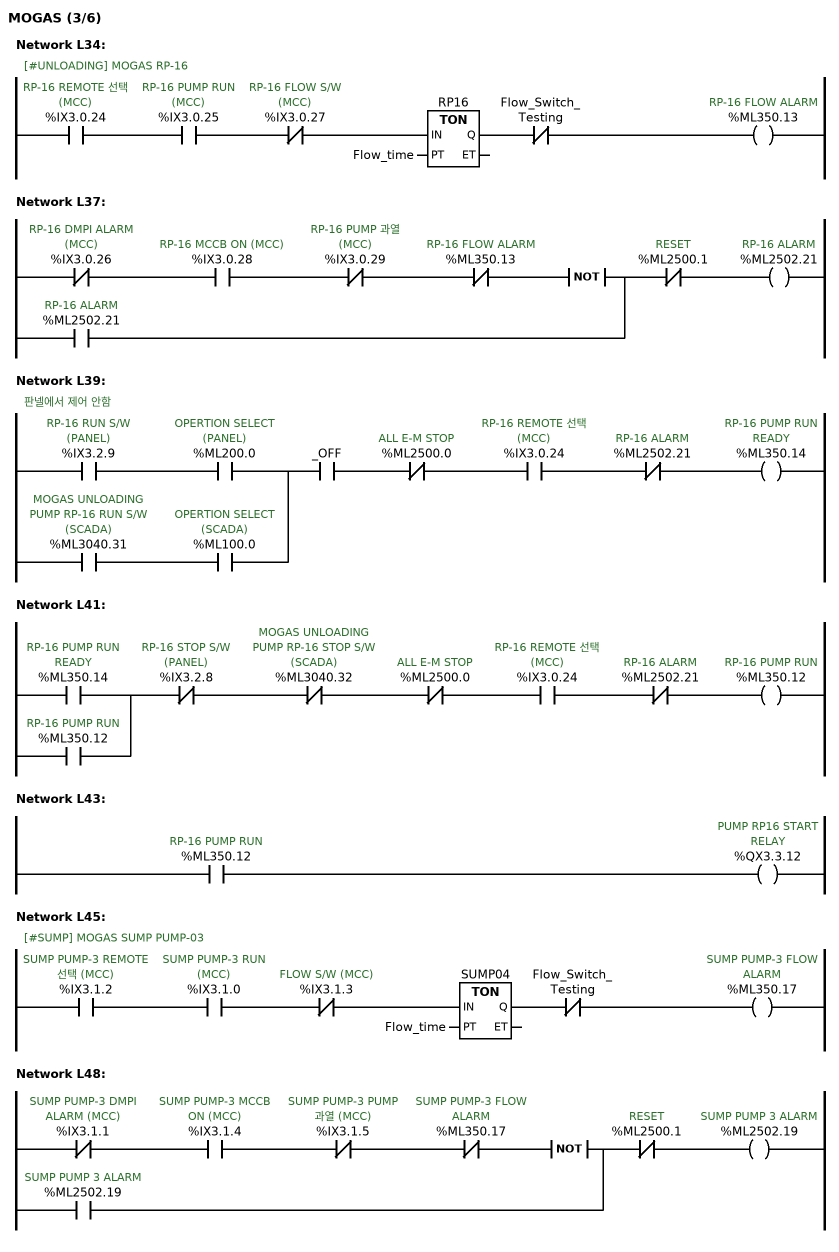
(* [#UNLOADING] MOGAS RP-16 *)
(* Rung L34 *)
RP16(IN := %IX3.0.24 AND %IX3.0.25 AND NOT %IX3.0.27, PT := Flow_time);
%ML350.13 := RP16.Q AND NOT Flow_Switch_Testing;
(* Rung L37 *)
%ML2502.21 := (NOT (NOT %IX3.0.26 AND %IX3.0.28 AND NOT %IX3.0.29 AND NOT %ML350.13) OR %ML2502.21) AND NOT %ML2500.1;
(* Rung L39 *)
%ML350.14 := ((%IX3.2.9 AND %ML200.0) OR (%ML3040.31 AND %ML100.0)) AND _OFF AND NOT %ML2500.0 AND %IX3.0.24 AND NOT %ML2502.21;
(* 판넬에서 제어 안함 *)
(* Rung L41 *)
%ML350.12 := (%ML350.14 OR %ML350.12) AND NOT %IX3.2.8 AND NOT %ML3040.32 AND NOT %ML2500.0 AND %IX3.0.24 AND NOT %ML2502.21;
(* Rung L43 *)
%QX3.3.12 := %ML350.12;
(* [#SUMP] MOGAS SUMP PUMP-03 *)
(* Rung L45 *)
SUMP04(IN := %IX3.1.2 AND %IX3.1.0 AND NOT %IX3.1.3, PT := Flow_time);
%ML350.17 := SUMP04.Q AND NOT Flow_Switch_Testing;
(* Rung L48 *)
%ML2502.19 := (NOT (NOT %IX3.1.1 AND %IX3.1.4 AND NOT %IX3.1.5 AND NOT %ML350.17) OR %ML2502.19) AND NOT %ML2500.1;

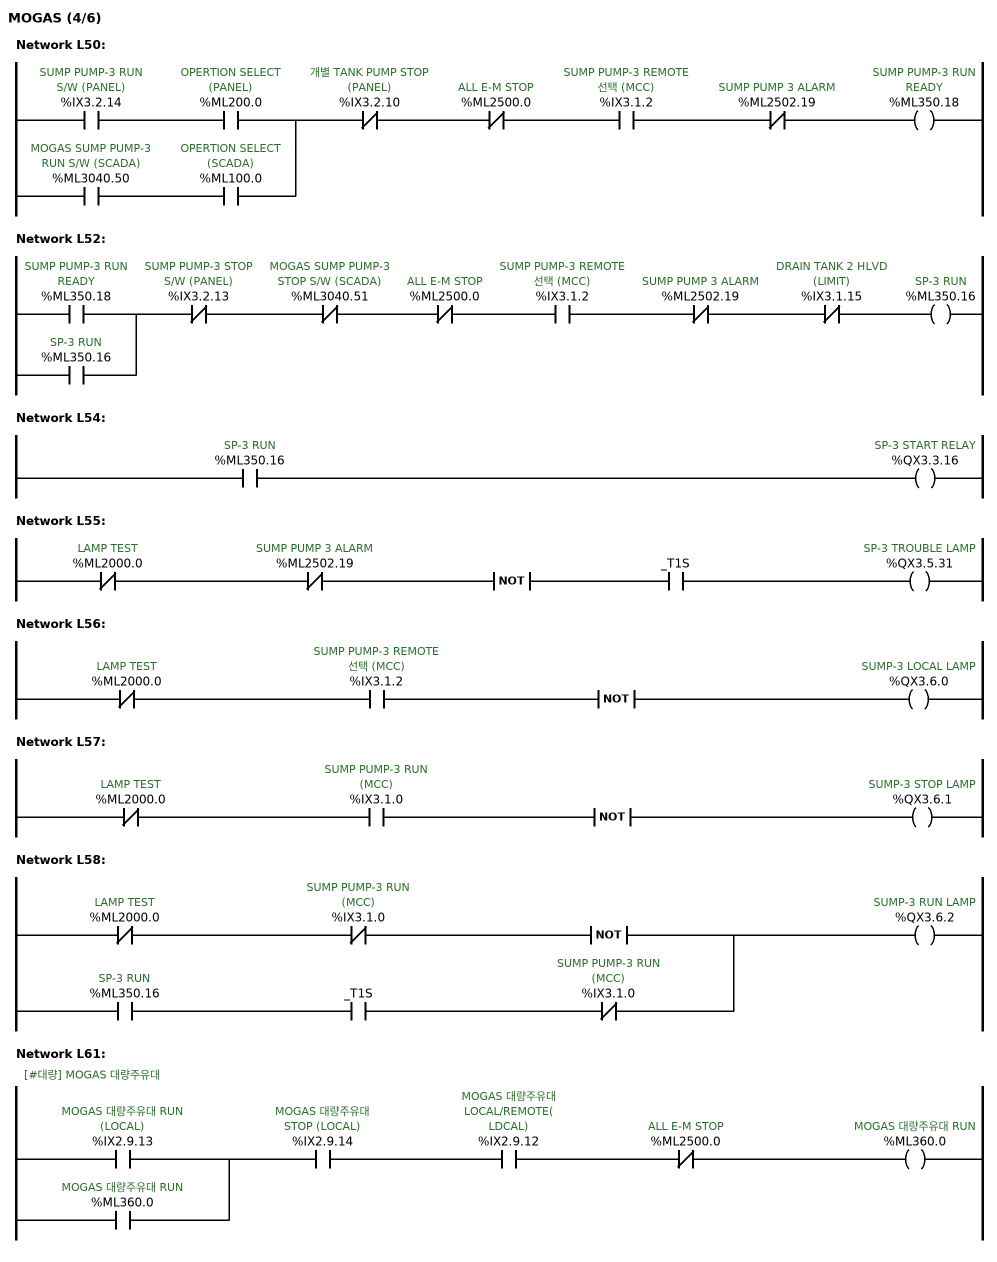
(* Rung L50 *)
%ML350.18 := ((%IX3.2.14 AND %ML200.0) OR (%ML3040.50 AND %ML100.0)) AND NOT %IX3.2.10 AND NOT %ML2500.0 AND %IX3.1.2 AND NOT %ML2502.19;
(* Rung L52 *)
%ML350.16 := (%ML350.18 OR %ML350.16) AND NOT %IX3.2.13 AND NOT %ML3040.51 AND NOT %ML2500.0 AND %IX3.1.2 AND NOT %ML2502.19 AND NOT %IX3.1.15;
(* Rung L54 *)
%QX3.3.16 := %ML350.16;
(* Rung L55 *)
%QX3.5.31 := NOT (NOT %ML2000.0 AND NOT %ML2502.19) AND _T1S;
(* Rung L56 *)
%QX3.6.0 := NOT (NOT %ML2000.0 AND %IX3.1.2);
(* Rung L57 *)
%QX3.6.1 := NOT (NOT %ML2000.0 AND %IX3.1.0);
(* Rung L58 *)
%QX3.6.2 := NOT (NOT %ML2000.0 AND NOT %IX3.1.0) OR (%ML350.16 AND _T1S AND NOT %IX3.1.0);
(* [#대량] MOGAS 대량주유대 *)
(* Rung L61 *)
%ML360.0 := (%IX2.9.13 OR %ML360.0) AND %IX2.9.14 AND %IX2.9.12 AND NOT %ML2500.0;

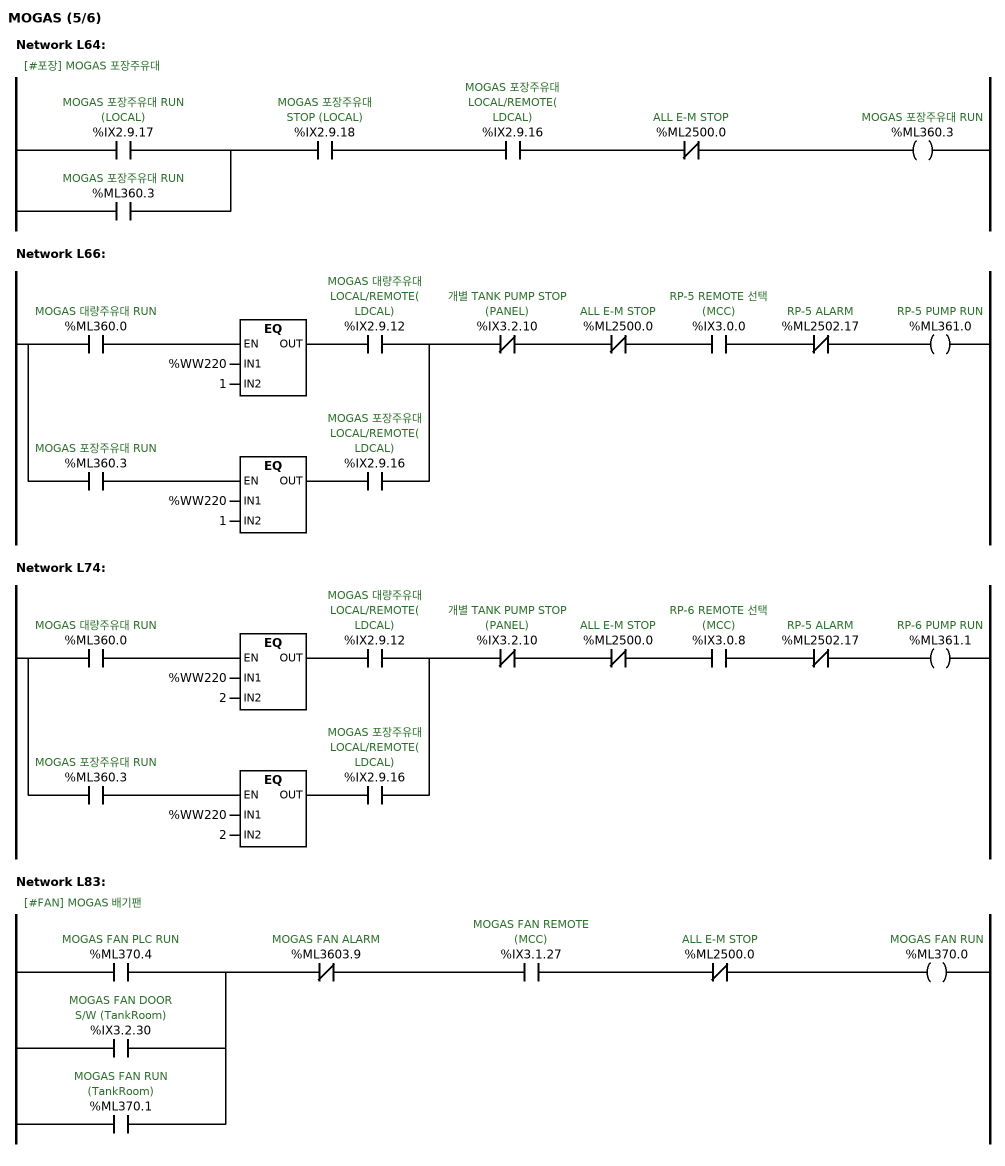
(* [#포장] MOGAS 포장주유대 *)
(* Rung L64 *)
%ML360.3 := (%IX2.9.17 OR %ML360.3) AND %IX2.9.18 AND %IX2.9.16 AND NOT %ML2500.0;
(* Rung L66 *)
IF %ML360.0 THEN _t1 := %WW220 = 1; END_IF;
IF %ML360.3 THEN _t2 := %WW220 = 1; END_IF;
%ML361.0 := ((_t1 AND %IX2.9.12) OR (_t2 AND %IX2.9.16)) AND NOT %IX3.2.10 AND NOT %ML2500.0 AND %IX3.0.0 AND NOT %ML2502.17;
(* Rung L74 *)
IF %ML360.0 THEN _t3 := %WW220 = 2; END_IF;
IF %ML360.3 THEN _t4 := %WW220 = 2; END_IF;
%ML361.1 := ((_t3 AND %IX2.9.12) OR (_t4 AND %IX2.9.16)) AND NOT %IX3.2.10 AND NOT %ML2500.0 AND %IX3.0.8 AND NOT %ML2502.17;
(* [#FAN] MOGAS 배기팬 *)
(* Rung L83 *)
%ML370.0 := (%ML370.4 OR %IX3.2.30 OR %ML370.1) AND NOT %ML3603.9 AND %IX3.1.27 AND NOT %ML2500.0;

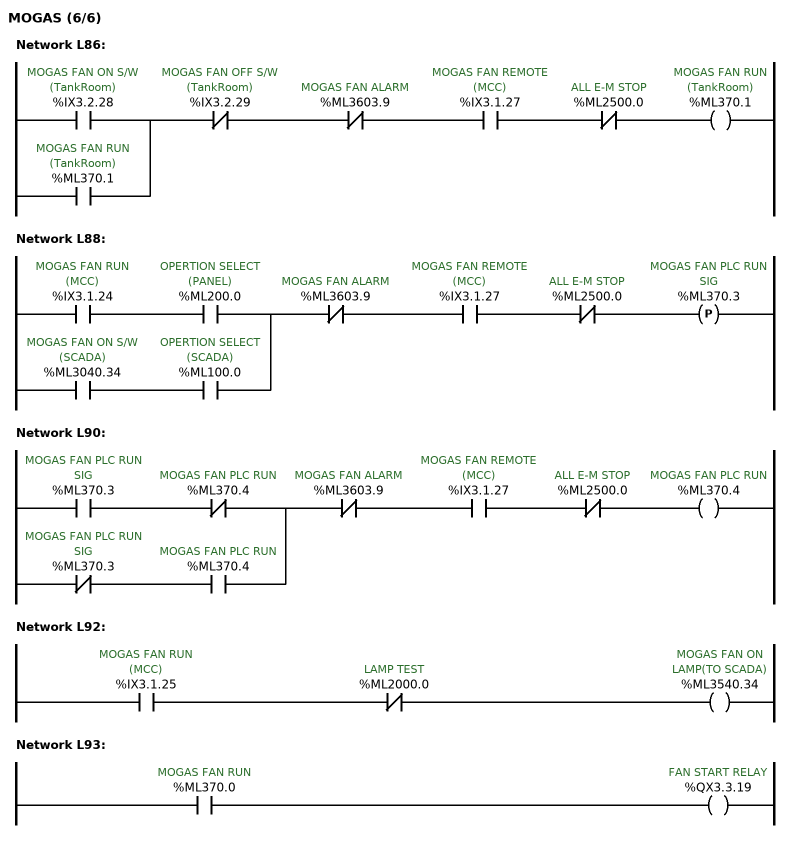
(* Rung L86 *)
%ML370.1 := (%IX3.2.28 OR %ML370.1) AND NOT %IX3.2.29 AND NOT %ML3603.9 AND %IX3.1.27 AND NOT %ML2500.0;
(* Rung L88 *)
_e5(CLK := ((%IX3.1.24 AND %ML200.0) OR (%ML3040.34 AND %ML100.0)) AND NOT %ML3603.9 AND %IX3.1.27 AND NOT %ML2500.0);
%ML370.3 := _e5.Q;
(* Rung L90 *)
%ML370.4 := ((%ML370.3 AND NOT %ML370.4) OR (NOT %ML370.3 AND %ML370.4)) AND NOT %ML3603.9 AND %IX3.1.27 AND NOT %ML2500.0;
(* Rung L92 *)
%ML3540.34 := %IX3.1.25 AND NOT %ML2000.0;
(* Rung L93 *)
%QX3.3.19 := %ML370.0;
END_PROGRAM

PROGRAM ANALOGUE (* task: 스캔 프로그램 *)
VAR
    DF1A_LEVEL_PER : INT;
    DF1B_LEVEL_PER : INT;
    DFM_LEVEL_PER : INT;
    DTK1_LEVEL_PER : INT;
    DTK2_LEVEL_PER : INT;
    FIT_1 : INT;
    FIT_2 : INT;
    MOGAS_LEVEL_PER : INT;
END_VAR
VAR_EXTERNAL
    _0108_CH0_ACT : BOOL; (* AT %UX1.8.16 *) (* 절연형 아날로그입력 모듈: 채널0 운전중 *)
    _0108_CH0_DATA : INT; (* AT %UW1.8.2 *) (* 절연형 아날로그입력 모듈: 채널0 변환값 *)
    _0108_CH0_IDD : BOOL; (* AT %UX1.8.160 *) (* 절연형 아날로그입력 모듈: 채널0 입력단선검출 *)
    _0108_CH1_ACT : BOOL; (* AT %UX1.8.17 *) (* 절연형 아날로그입력 모듈: 채널1 운전중 *)
    _0108_CH1_DATA : INT; (* AT %UW1.8.3 *) (* 절연형 아날로그입력 모듈: 채널1 변환값 *)
    _0108_CH1_IDD : BOOL; (* AT %UX1.8.161 *) (* 절연형 아날로그입력 모듈: 채널1 입력단선검출 *)
    _0108_CH2_ACT : BOOL; (* AT %UX1.8.18 *) (* 절연형 아날로그입력 모듈: 채널2 운전중 *)
    _0108_CH2_DATA : INT; (* AT %UW1.8.4 *) (* 절연형 아날로그입력 모듈: 채널2 변환값 *)
    _0108_CH2_IDD : BOOL; (* AT %UX1.8.162 *) (* 절연형 아날로그입력 모듈: 채널2 입력단선검출 *)
    _0108_CH3_ACT : BOOL; (* AT %UX1.8.19 *) (* 절연형 아날로그입력 모듈: 채널3 운전중 *)
    _0108_CH3_DATA : INT; (* AT %UW1.8.5 *) (* 절연형 아날로그입력 모듈: 채널3 변환값 *)
    _0108_CH3_IDD : BOOL; (* AT %UX1.8.163 *) (* 절연형 아날로그입력 모듈: 채널3 입력단선검출 *)
    _0109_CH0_ACT : BOOL; (* AT %UX1.9.16 *) (* 절연형 아날로그출력 모듈: 채널0 운전중 *)
    _0109_CH0_DATA : INT; (* AT %UW1.9.3 *) (* 절연형 아날로그출력 모듈: 채널0 입력값 *)
    _0109_CH0_ERR : BOOL; (* AT %UX1.9.0 *) (* 절연형 아날로그출력 모듈: 채널0 에러 *)
    _0109_CH0_OUTEN : BOOL; (* AT %UX1.9.32 *) (* 절연형 아날로그출력 모듈: 채널0 출력상태설정 *)
    _0109_CH1_ACT : BOOL; (* AT %UX1.9.17 *) (* 절연형 아날로그출력 모듈: 채널1 운전중 *)
    _0109_CH1_DATA : INT; (* AT %UW1.9.4 *) (* 절연형 아날로그출력 모듈: 채널1 입력값 *)
    _0109_CH1_ERR : BOOL; (* AT %UX1.9.1 *) (* 절연형 아날로그출력 모듈: 채널1 에러 *)
    _0109_CH2_ACT : BOOL; (* AT %UX1.9.18 *) (* 절연형 아날로그출력 모듈: 채널2 운전중 *)
    _0109_CH2_DATA : INT; (* AT %UW1.9.5 *) (* 절연형 아날로그출력 모듈: 채널2 입력값 *)
    _0109_CH2_ERR : BOOL; (* AT %UX1.9.2 *) (* 절연형 아날로그출력 모듈: 채널2 에러 *)
    _0109_CH3_ACT : BOOL; (* AT %UX1.9.19 *) (* 절연형 아날로그출력 모듈: 채널3 운전중 *)
    _0109_CH3_DATA : INT; (* AT %UW1.9.6 *) (* 절연형 아날로그출력 모듈: 채널3 입력값 *)
    _0109_CH3_ERR : BOOL; (* AT %UX1.9.3 *) (* 절연형 아날로그출력 모듈: 채널3 에러 *)
    _0109_OUTEN : WORD; (* AT %UW1.9.2 *) (* 절연형 아날로그출력 모듈: 출력상태 설정 *)
    _0110_CH0_ACT : BOOL; (* AT %UX1.10.16 *) (* 절연형 아날로그출력 모듈: 채널0 운전중 *)
    _0110_CH0_DATA : INT; (* AT %UW1.10.3 *) (* 절연형 아날로그출력 모듈: 채널0 입력값 *)
    _0110_CH0_ERR : BOOL; (* AT %UX1.10.0 *) (* 절연형 아날로그출력 모듈: 채널0 에러 *)
    _0110_OUTEN : WORD; (* AT %UW1.10.2 *) (* 절연형 아날로그출력 모듈: 출력상태 설정 *)
    _0206_CH0_ACT : BOOL; (* AT %UX2.6.16 *) (* 절연형 아날로그입력 모듈: 채널0 운전중 *)
    _0206_CH0_DATA : INT; (* AT %UW2.6.2 *) (* 절연형 아날로그입력 모듈: 채널0 변환값 *)
    _0206_CH0_IDD : BOOL; (* AT %UX2.6.160 *) (* 절연형 아날로그입력 모듈: 채널0 입력단선검출 *)
    _0206_CH1_ACT : BOOL; (* AT %UX2.6.17 *) (* 절연형 아날로그입력 모듈: 채널1 운전중 *)
    _0206_CH1_DATA : INT; (* AT %UW2.6.3 *) (* 절연형 아날로그입력 모듈: 채널1 변환값 *)
    _0206_CH1_IDD : BOOL; (* AT %UX2.6.161 *) (* 절연형 아날로그입력 모듈: 채널1 입력단선검출 *)
    _0206_CH2_ACT : BOOL; (* AT %UX2.6.18 *) (* 절연형 아날로그입력 모듈: 채널2 운전중 *)
    _0206_CH2_DATA : INT; (* AT %UW2.6.4 *) (* 절연형 아날로그입력 모듈: 채널2 변환값 *)
    _0206_CH2_IDD : BOOL; (* AT %UX2.6.162 *) (* 절연형 아날로그입력 모듈: 채널2 입력단선검출 *)
    _0206_CH3_ACT : BOOL; (* AT %UX2.6.19 *) (* 절연형 아날로그입력 모듈: 채널3 운전중 *)
    _0206_CH3_DATA : INT; (* AT %UW2.6.5 *) (* 절연형 아날로그입력 모듈: 채널3 변환값 *)
    _0206_CH3_IDD : BOOL; (* AT %UX2.6.163 *) (* 절연형 아날로그입력 모듈: 채널3 입력단선검출 *)
    _0207_CH0_ACT : BOOL; (* AT %UX2.7.16 *) (* 절연형 아날로그출력 모듈: 채널0 운전중 *)
    _0207_CH0_DATA : INT; (* AT %UW2.7.3 *) (* 절연형 아날로그출력 모듈: 채널0 입력값 *)
    _0207_CH0_ERR : BOOL; (* AT %UX2.7.0 *) (* 절연형 아날로그출력 모듈: 채널0 에러 *)
    _0207_CH1_ACT : BOOL; (* AT %UX2.7.17 *) (* 절연형 아날로그출력 모듈: 채널1 운전중 *)
    _0207_CH1_DATA : INT; (* AT %UW2.7.4 *) (* 절연형 아날로그출력 모듈: 채널1 입력값 *)
    _0207_CH2_ACT : BOOL; (* AT %UX2.7.18 *) (* 절연형 아날로그출력 모듈: 채널2 운전중 *)
    _0207_CH2_DATA : INT; (* AT %UW2.7.5 *) (* 절연형 아날로그출력 모듈: 채널2 입력값 *)
    _0207_CH2_ERR : BOOL; (* AT %UX2.7.2 *) (* 절연형 아날로그출력 모듈: 채널2 에러 *)
    _0207_CH3_DATA : INT; (* AT %UW2.7.6 *) (* 절연형 아날로그출력 모듈: 채널3 입력값 *)
    _0207_OUTEN : WORD; (* AT %UW2.7.2 *) (* 절연형 아날로그출력 모듈: 출력상태 설정 *)
    _0307_CH0_ACT : BOOL; (* AT %UX3.7.16 *) (* 절연형 아날로그입력 모듈: 채널0 운전중 *)
    _0307_CH0_DATA : INT; (* AT %UW3.7.2 *) (* 절연형 아날로그입력 모듈: 채널0 변환값 *)
    _0307_CH0_IDD : BOOL; (* AT %UX3.7.160 *) (* 절연형 아날로그입력 모듈: 채널0 입력단선검출 *)
    _0307_CH1_ACT : BOOL; (* AT %UX3.7.17 *) (* 절연형 아날로그입력 모듈: 채널1 운전중 *)
    _0307_CH1_DATA : INT; (* AT %UW3.7.3 *) (* 절연형 아날로그입력 모듈: 채널1 변환값 *)
    _0307_CH1_IDD : BOOL; (* AT %UX3.7.161 *) (* 절연형 아날로그입력 모듈: 채널1 입력단선검출 *)
    _0307_CH2_ACT : BOOL; (* AT %UX3.7.18 *) (* 절연형 아날로그입력 모듈: 채널2 운전중 *)
    _0307_CH2_DATA : INT; (* AT %UW3.7.4 *) (* 절연형 아날로그입력 모듈: 채널2 변환값 *)
    _0307_CH2_IDD : BOOL; (* AT %UX3.7.162 *) (* 절연형 아날로그입력 모듈: 채널2 입력단선검출 *)
    _0307_CH3_DATA : INT; (* AT %UW3.7.5 *) (* 절연형 아날로그입력 모듈: 채널3 변환값 *)
    _0307_CH3_IDD : BOOL; (* AT %UX3.7.163 *) (* 절연형 아날로그입력 모듈: 채널3 입력단선검출 *)
    _0308_CH0_ACT : BOOL; (* AT %UX3.8.16 *) (* 절연형 아날로그출력 모듈: 채널0 운전중 *)
    _0308_CH0_DATA : INT; (* AT %UW3.8.3 *) (* 절연형 아날로그출력 모듈: 채널0 입력값 *)
    _0308_CH1_ACT : BOOL; (* AT %UX3.8.17 *) (* 절연형 아날로그출력 모듈: 채널1 운전중 *)
    _0308_CH1_DATA : INT; (* AT %UW3.8.4 *) (* 절연형 아날로그출력 모듈: 채널1 입력값 *)
    _0308_CH2_ACT : BOOL; (* AT %UX3.8.18 *) (* 절연형 아날로그출력 모듈: 채널2 운전중 *)
    _0308_CH2_DATA : INT; (* AT %UW3.8.5 *) (* 절연형 아날로그출력 모듈: 채널2 입력값 *)
    _0308_CH2_ERR : BOOL; (* AT %UX3.8.2 *) (* 절연형 아날로그출력 모듈: 채널2 에러 *)
    _0308_CH3_ACT : BOOL; (* AT %UX3.8.19 *) (* 절연형 아날로그출력 모듈: 채널3 운전중 *)
    _0308_CH3_DATA : INT; (* AT %UW3.8.6 *) (* 절연형 아날로그출력 모듈: 채널3 입력값 *)
    _0308_CH3_ERR : BOOL; (* AT %UX3.8.3 *) (* 절연형 아날로그출력 모듈: 채널3 에러 *)
    _0308_OUTEN : WORD; (* AT %UW3.8.2 *) (* 절연형 아날로그출력 모듈: 출력상태 설정 *)
END_VAR
VAR_EXTERNAL CONSTANT
    _F0308_CH0_DEC_RATE : UINT; (* 절연형 아날로그출력 모듈: 채널0 변화율 감소값 *)
    _F0308_CH0_STAT : UINT; (* 절연형 아날로그출력 모듈: 채널0 이상 상태 출력 설정값 *)
    _F0308_LIMIT_EN : UINT; (* 절연형 아날로그출력 모듈: 출력제한 채널 설정 *)
END_VAR
VAR
    _t1 : BOOL;
    _t2 : BOOL;
    _t3 : BOOL;
    _t4 : BOOL;
    _t5 : BOOL;
    _t6 : BOOL;
    _t7 : BOOL;
    _t8 : BOOL;
    _t9 : BOOL;
    _t10 : BOOL;
    _t11 : BOOL;
    _t12 : BOOL;
    _t13 : BOOL;
END_VAR

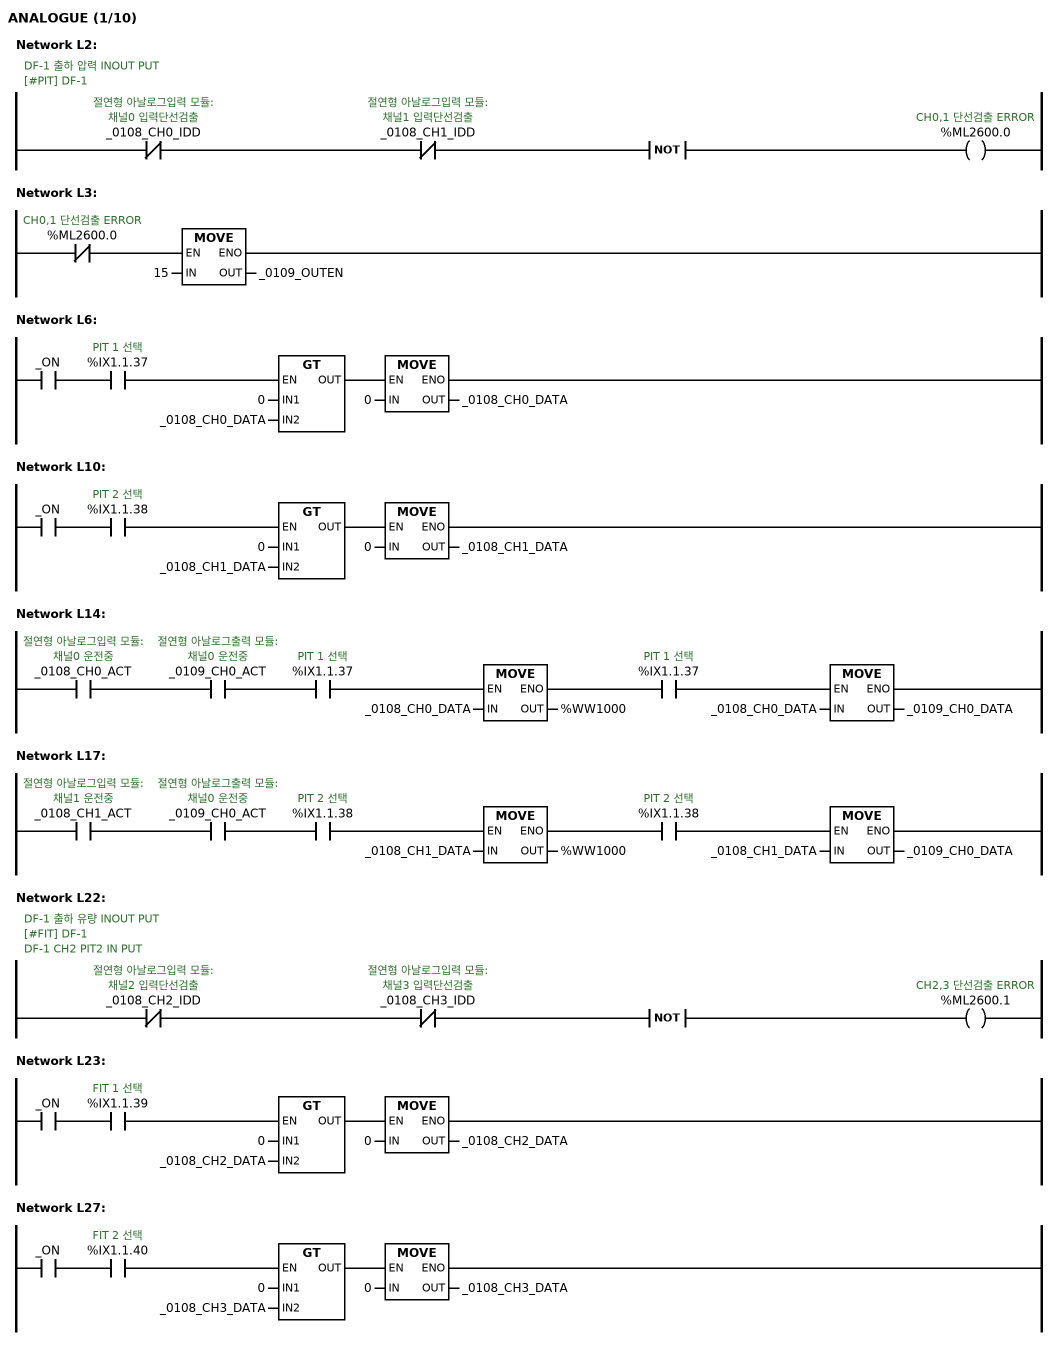
(* DF-1 출하 압력 INOUT PUT *)
(* [#PIT] DF-1 *)
(* Rung L2 *)
%ML2600.0 := NOT (NOT _0108_CH0_IDD AND NOT _0108_CH1_IDD);
(*  *)
(* Rung L3 *)
IF NOT %ML2600.0 THEN _0109_OUTEN := 15; END_IF;
(* Rung L6 *)
IF _ON AND %IX1.1.37 THEN _t1 := 0 > _0108_CH0_DATA; END_IF;
IF _t1 THEN _0108_CH0_DATA := 0; END_IF;
(* Rung L10 *)
IF _ON AND %IX1.1.38 THEN _t2 := 0 > _0108_CH1_DATA; END_IF;
IF _t2 THEN _0108_CH1_DATA := 0; END_IF;
(* Rung L14 *)
IF _0108_CH0_ACT AND _0109_CH0_ACT AND %IX1.1.37 THEN %WW1000 := _0108_CH0_DATA; END_IF;
IF _0108_CH0_ACT AND _0109_CH0_ACT AND %IX1.1.37 AND %IX1.1.37 THEN
    _0109_CH0_DATA := _0108_CH0_DATA;
END_IF;
(* Rung L17 *)
IF _0108_CH1_ACT AND _0109_CH0_ACT AND %IX1.1.38 THEN %WW1000 := _0108_CH1_DATA; END_IF;
IF _0108_CH1_ACT AND _0109_CH0_ACT AND %IX1.1.38 AND %IX1.1.38 THEN
    _0109_CH0_DATA := _0108_CH1_DATA;
END_IF;
(* DF-1 출하 유량 INOUT PUT *)
(* [#FIT] DF-1 *)
(* Rung L22 *)
%ML2600.1 := NOT (NOT _0108_CH2_IDD AND NOT _0108_CH3_IDD);
(* DF-1 CH2 PIT2 IN PUT *)
(* Rung L23 *)
IF _ON AND %IX1.1.39 THEN _t3 := 0 > _0108_CH2_DATA; END_IF;
IF _t3 THEN _0108_CH2_DATA := 0; END_IF;
(* Rung L27 *)
IF _ON AND %IX1.1.40 THEN _t4 := 0 > _0108_CH3_DATA; END_IF;
IF _t4 THEN _0108_CH3_DATA := 0; END_IF;

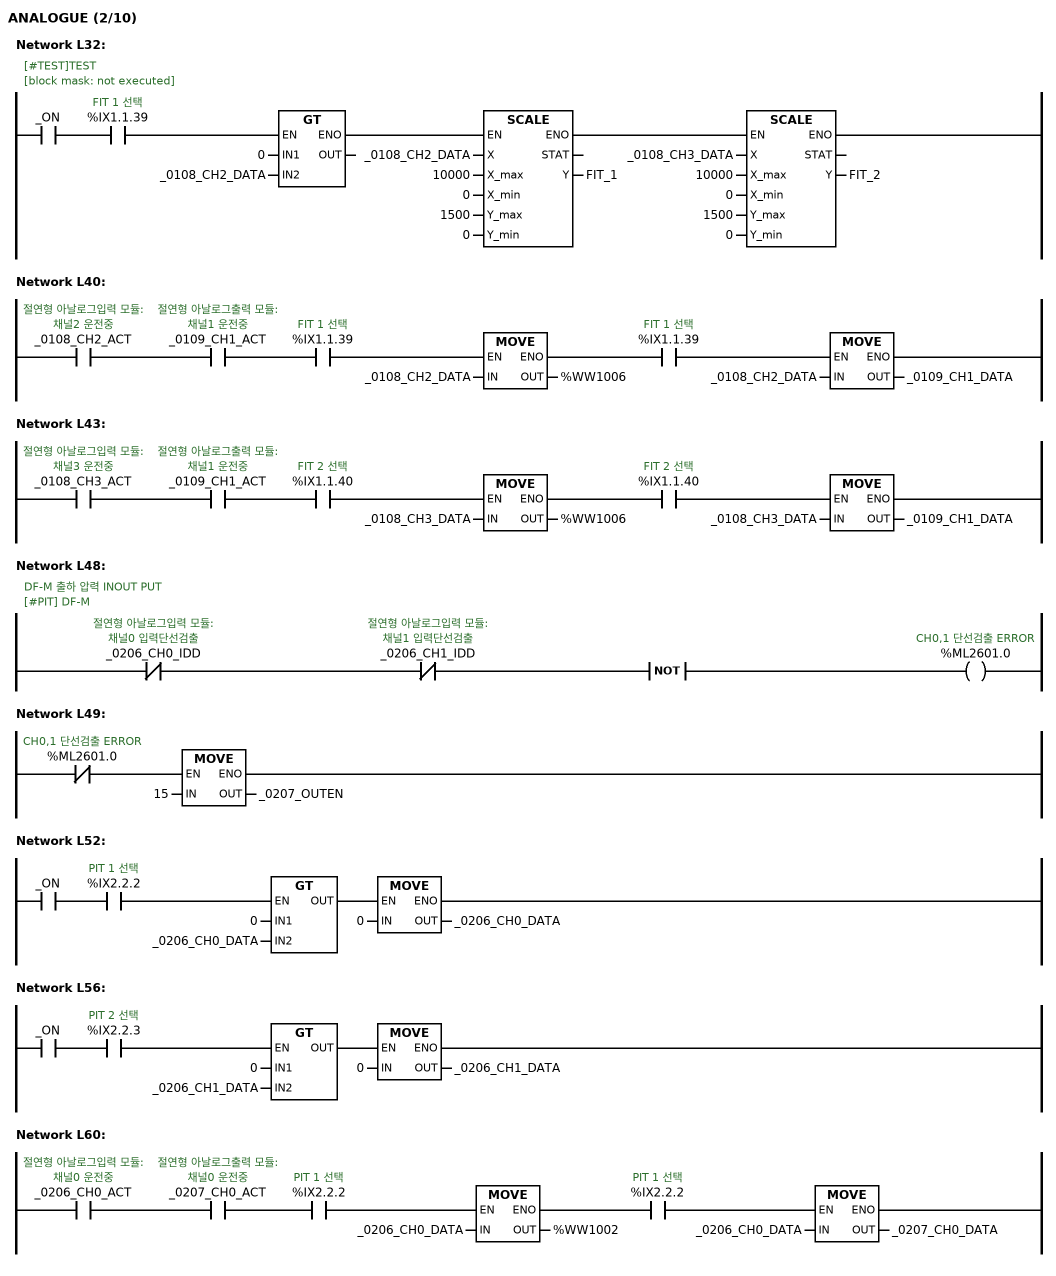
(* [#TEST]TEST *)
(* Rung L32 is block-masked: not executed *)
// IF _ON AND %IX1.1.39 THEN
//     _t5 := 0 > _0108_CH2_DATA;
//     SCALE(X := _0108_CH2_DATA, X_max := 10000, X_min := 0, Y_max := 1500, Y_min := 0, Y => FIT_1);
//     SCALE(X := _0108_CH3_DATA, X_max := 10000, X_min := 0, Y_max := 1500, Y_min := 0, Y => FIT_2);
// END_IF;
(*  *)
(* Rung L40 *)
IF _0108_CH2_ACT AND _0109_CH1_ACT AND %IX1.1.39 THEN %WW1006 := _0108_CH2_DATA; END_IF;
IF _0108_CH2_ACT AND _0109_CH1_ACT AND %IX1.1.39 AND %IX1.1.39 THEN
    _0109_CH1_DATA := _0108_CH2_DATA;
END_IF;
(* Rung L43 *)
IF _0108_CH3_ACT AND _0109_CH1_ACT AND %IX1.1.40 THEN %WW1006 := _0108_CH3_DATA; END_IF;
IF _0108_CH3_ACT AND _0109_CH1_ACT AND %IX1.1.40 AND %IX1.1.40 THEN
    _0109_CH1_DATA := _0108_CH3_DATA;
END_IF;
(* DF-M 출하 압력 INOUT PUT *)
(* [#PIT] DF-M *)
(* Rung L48 *)
%ML2601.0 := NOT (NOT _0206_CH0_IDD AND NOT _0206_CH1_IDD);
(*  *)
(* Rung L49 *)
IF NOT %ML2601.0 THEN _0207_OUTEN := 15; END_IF;
(* Rung L52 *)
IF _ON AND %IX2.2.2 THEN _t6 := 0 > _0206_CH0_DATA; END_IF;
IF _t6 THEN _0206_CH0_DATA := 0; END_IF;
(* Rung L56 *)
IF _ON AND %IX2.2.3 THEN _t7 := 0 > _0206_CH1_DATA; END_IF;
IF _t7 THEN _0206_CH1_DATA := 0; END_IF;
(* Rung L60 *)
IF _0206_CH0_ACT AND _0207_CH0_ACT AND %IX2.2.2 THEN %WW1002 := _0206_CH0_DATA; END_IF;
IF _0206_CH0_ACT AND _0207_CH0_ACT AND %IX2.2.2 AND %IX2.2.2 THEN
    _0207_CH0_DATA := _0206_CH0_DATA;
END_IF;

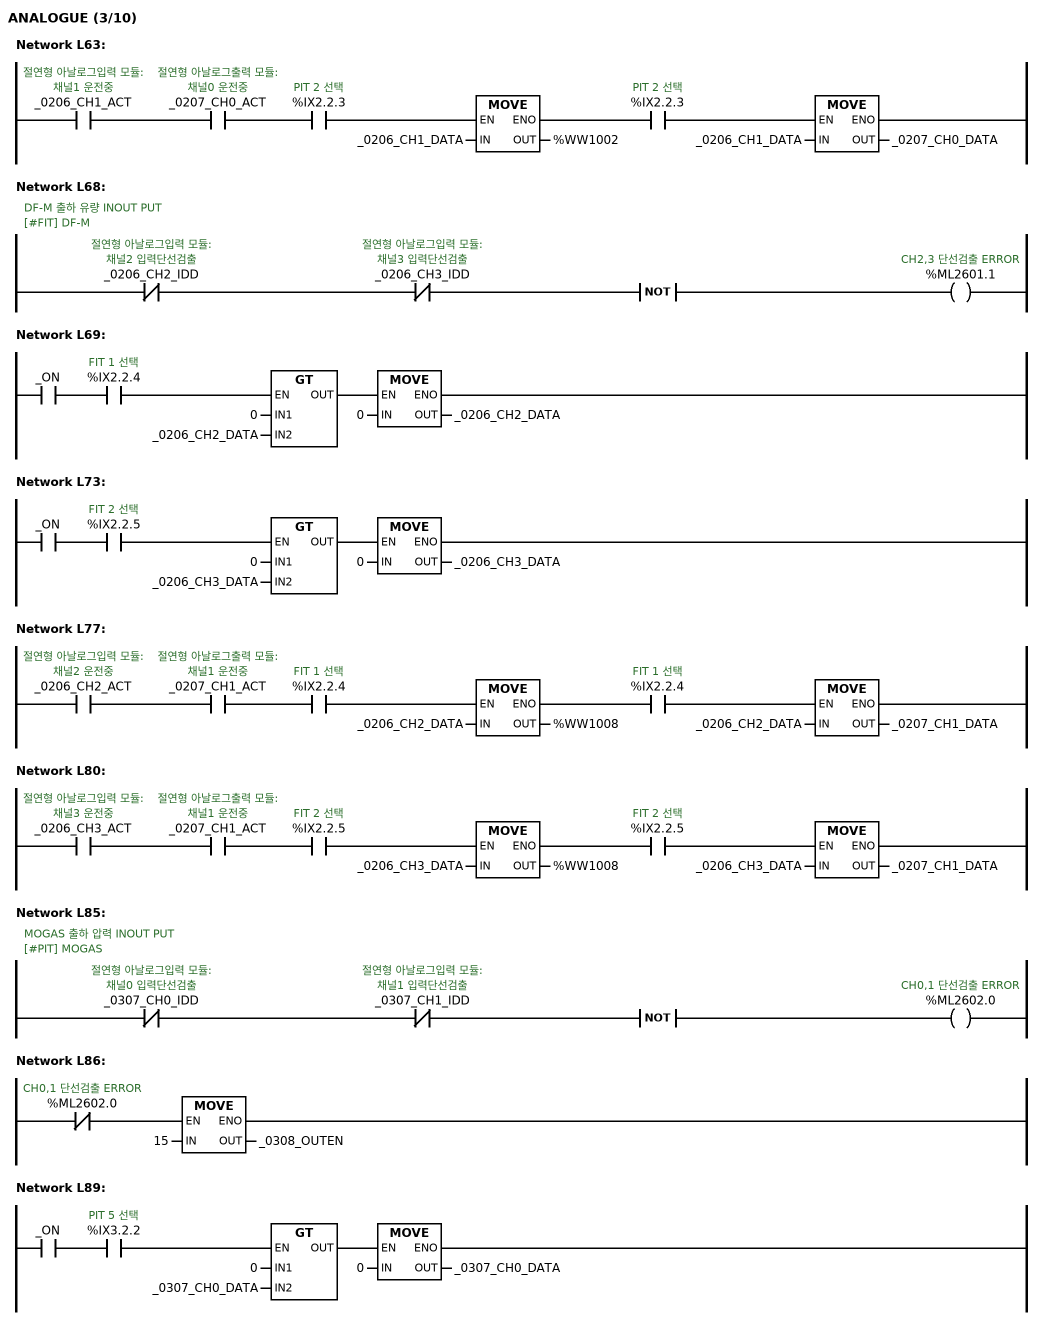
(* Rung L63 *)
IF _0206_CH1_ACT AND _0207_CH0_ACT AND %IX2.2.3 THEN %WW1002 := _0206_CH1_DATA; END_IF;
IF _0206_CH1_ACT AND _0207_CH0_ACT AND %IX2.2.3 AND %IX2.2.3 THEN
    _0207_CH0_DATA := _0206_CH1_DATA;
END_IF;
(* DF-M 출하 유량 INOUT PUT *)
(* [#FIT] DF-M *)
(* Rung L68 *)
%ML2601.1 := NOT (NOT _0206_CH2_IDD AND NOT _0206_CH3_IDD);
(*  *)
(* Rung L69 *)
IF _ON AND %IX2.2.4 THEN _t8 := 0 > _0206_CH2_DATA; END_IF;
IF _t8 THEN _0206_CH2_DATA := 0; END_IF;
(* Rung L73 *)
IF _ON AND %IX2.2.5 THEN _t9 := 0 > _0206_CH3_DATA; END_IF;
IF _t9 THEN _0206_CH3_DATA := 0; END_IF;
(* Rung L77 *)
IF _0206_CH2_ACT AND _0207_CH1_ACT AND %IX2.2.4 THEN %WW1008 := _0206_CH2_DATA; END_IF;
IF _0206_CH2_ACT AND _0207_CH1_ACT AND %IX2.2.4 AND %IX2.2.4 THEN
    _0207_CH1_DATA := _0206_CH2_DATA;
END_IF;
(* Rung L80 *)
IF _0206_CH3_ACT AND _0207_CH1_ACT AND %IX2.2.5 THEN %WW1008 := _0206_CH3_DATA; END_IF;
IF _0206_CH3_ACT AND _0207_CH1_ACT AND %IX2.2.5 AND %IX2.2.5 THEN
    _0207_CH1_DATA := _0206_CH3_DATA;
END_IF;
(* MOGAS 출하 압력 INOUT PUT *)
(* [#PIT] MOGAS *)
(* Rung L85 *)
%ML2602.0 := NOT (NOT _0307_CH0_IDD AND NOT _0307_CH1_IDD);
(*  *)
(* Rung L86 *)
IF NOT %ML2602.0 THEN _0308_OUTEN := 15; END_IF;
(* Rung L89 *)
IF _ON AND %IX3.2.2 THEN _t10 := 0 > _0307_CH0_DATA; END_IF;
IF _t10 THEN _0307_CH0_DATA := 0; END_IF;

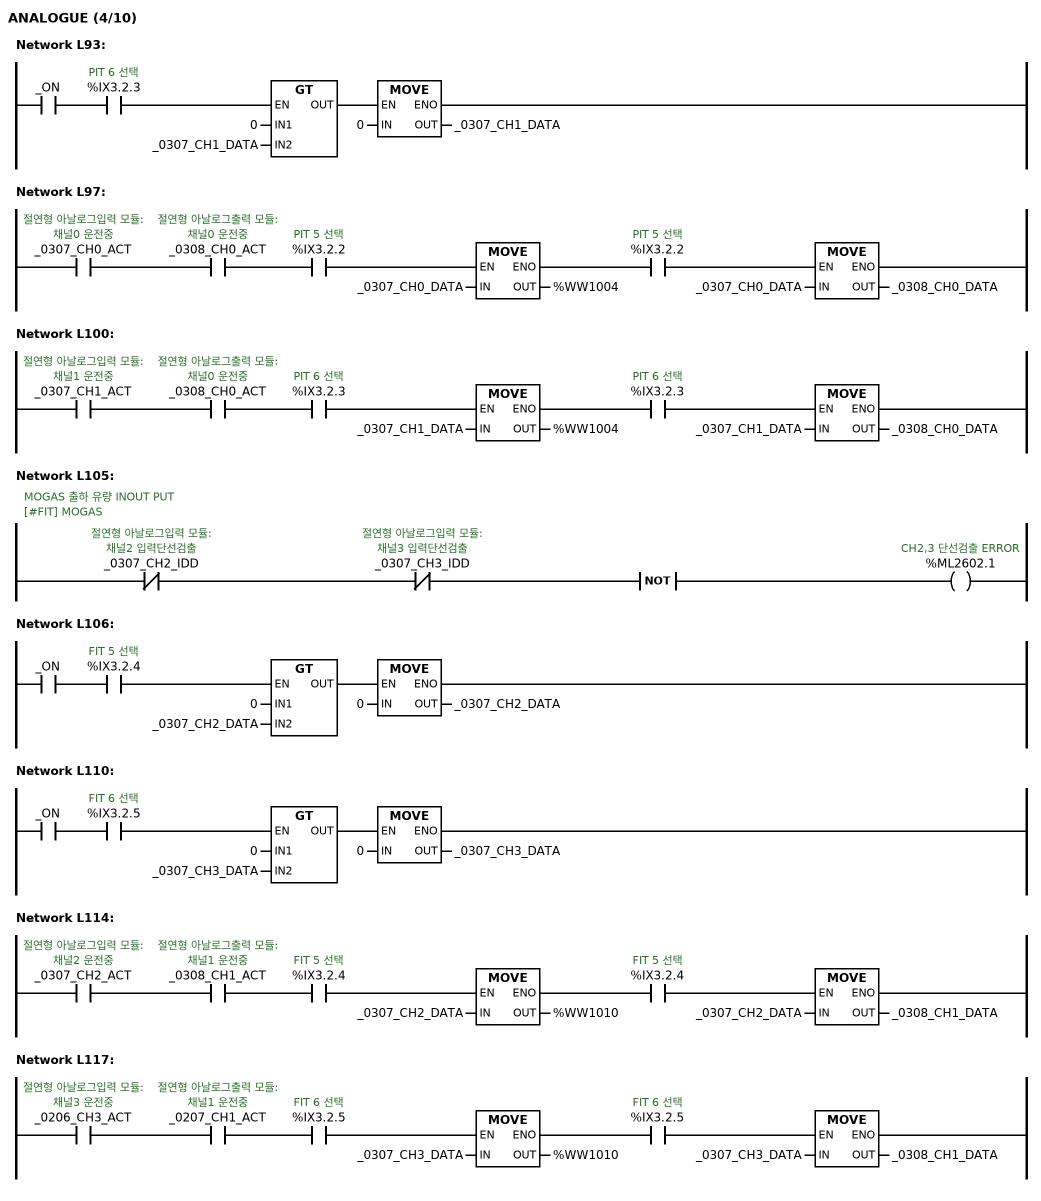
(* Rung L93 *)
IF _ON AND %IX3.2.3 THEN _t11 := 0 > _0307_CH1_DATA; END_IF;
IF _t11 THEN _0307_CH1_DATA := 0; END_IF;
(* Rung L97 *)
IF _0307_CH0_ACT AND _0308_CH0_ACT AND %IX3.2.2 THEN %WW1004 := _0307_CH0_DATA; END_IF;
IF _0307_CH0_ACT AND _0308_CH0_ACT AND %IX3.2.2 AND %IX3.2.2 THEN
    _0308_CH0_DATA := _0307_CH0_DATA;
END_IF;
(* Rung L100 *)
IF _0307_CH1_ACT AND _0308_CH0_ACT AND %IX3.2.3 THEN %WW1004 := _0307_CH1_DATA; END_IF;
IF _0307_CH1_ACT AND _0308_CH0_ACT AND %IX3.2.3 AND %IX3.2.3 THEN
    _0308_CH0_DATA := _0307_CH1_DATA;
END_IF;
(* MOGAS 출하 유량 INOUT PUT *)
(* [#FIT] MOGAS *)
(* Rung L105 *)
%ML2602.1 := NOT (NOT _0307_CH2_IDD AND NOT _0307_CH3_IDD);
(*  *)
(* Rung L106 *)
IF _ON AND %IX3.2.4 THEN _t12 := 0 > _0307_CH2_DATA; END_IF;
IF _t12 THEN _0307_CH2_DATA := 0; END_IF;
(* Rung L110 *)
IF _ON AND %IX3.2.5 THEN _t13 := 0 > _0307_CH3_DATA; END_IF;
IF _t13 THEN _0307_CH3_DATA := 0; END_IF;
(* Rung L114 *)
IF _0307_CH2_ACT AND _0308_CH1_ACT AND %IX3.2.4 THEN %WW1010 := _0307_CH2_DATA; END_IF;
IF _0307_CH2_ACT AND _0308_CH1_ACT AND %IX3.2.4 AND %IX3.2.4 THEN
    _0308_CH1_DATA := _0307_CH2_DATA;
END_IF;
(* Rung L117 *)
IF _0206_CH3_ACT AND _0207_CH1_ACT AND %IX3.2.5 THEN %WW1010 := _0307_CH3_DATA; END_IF;
IF _0206_CH3_ACT AND _0207_CH1_ACT AND %IX3.2.5 AND %IX3.2.5 THEN
    _0308_CH1_DATA := _0307_CH3_DATA;
END_IF;

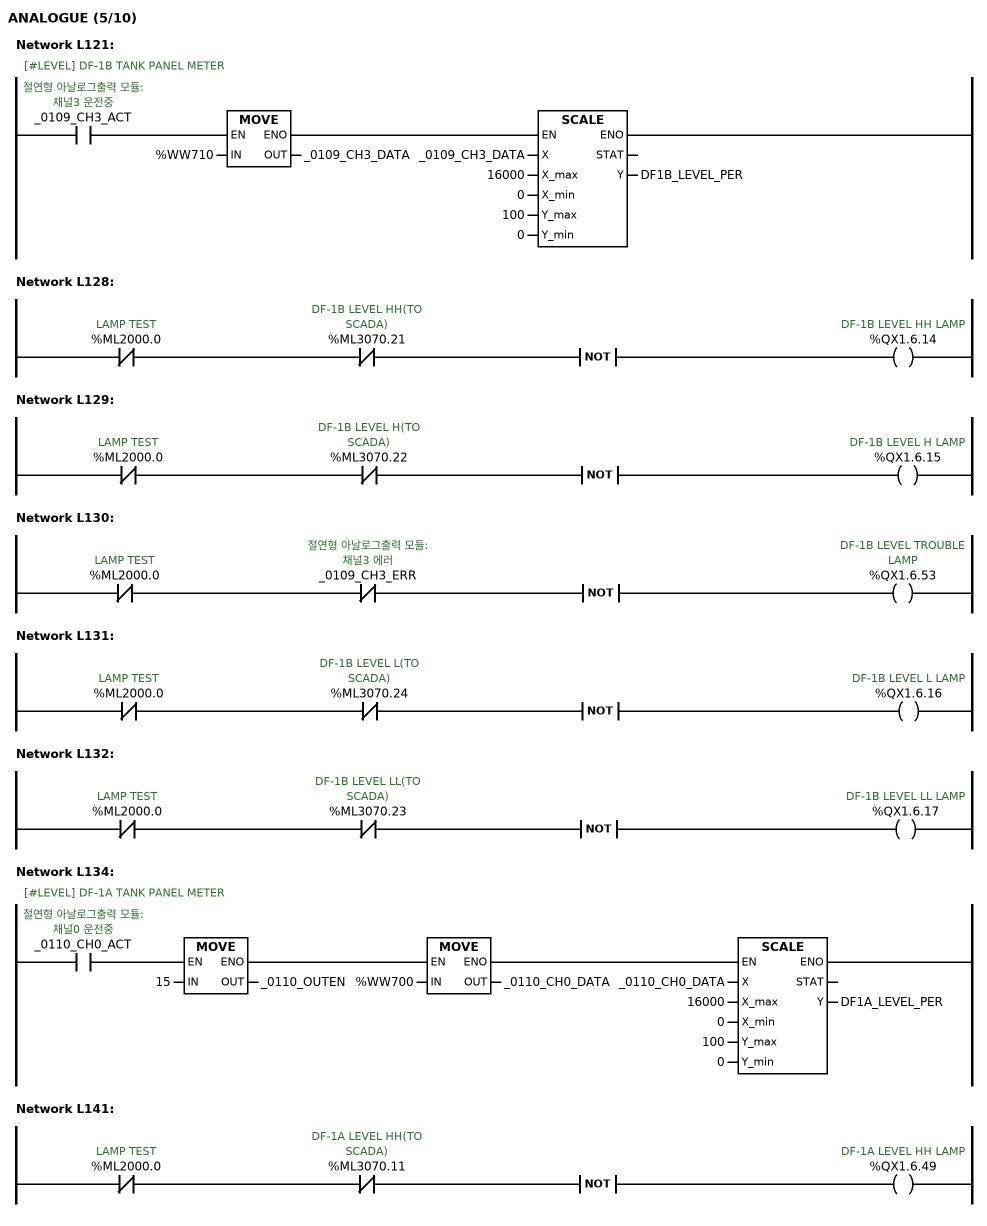
(* [#LEVEL] DF-1B TANK PANEL METER *)
(* Rung L121 *)
IF _0109_CH3_ACT THEN
    _0109_CH3_DATA := %WW710;
    SCALE(X := _0109_CH3_DATA, X_max := 16000, X_min := 0, Y_max := 100, Y_min := 0, Y => DF1B_LEVEL_PER);
END_IF;
(* Rung L128 *)
%QX1.6.14 := NOT (NOT %ML2000.0 AND NOT %ML3070.21);
(* Rung L129 *)
%QX1.6.15 := NOT (NOT %ML2000.0 AND NOT %ML3070.22);
(* Rung L130 *)
%QX1.6.53 := NOT (NOT %ML2000.0 AND NOT _0109_CH3_ERR);
(* Rung L131 *)
%QX1.6.16 := NOT (NOT %ML2000.0 AND NOT %ML3070.24);
(* Rung L132 *)
%QX1.6.17 := NOT (NOT %ML2000.0 AND NOT %ML3070.23);
(* [#LEVEL] DF-1A TANK PANEL METER *)
(* Rung L134 *)
IF _0110_CH0_ACT THEN
    _0110_OUTEN := 15;
    _0110_CH0_DATA := %WW700;
    SCALE(X := _0110_CH0_DATA, X_max := 16000, X_min := 0, Y_max := 100, Y_min := 0, Y => DF1A_LEVEL_PER);
END_IF;
(* Rung L141 *)
%QX1.6.49 := NOT (NOT %ML2000.0 AND NOT %ML3070.11);

